LIN {X 0,Y 418.225,Z 378.998,A -85,B 0,C 180,E1 -10215.107,E2 -10215.107} C_VEL
LIN {X 0,Y 418.208,Z 379.016,A -85,B 0,C 180,E1 -10217.763,E2 -10217.763} C_VEL
LIN {X 0,Y 418.223,Z 379.009,A -85,B 0,C 180,E1 -10221.555,E2 -10221.555} C_VEL
LIN {X 0,Y 418.238,Z 379.011,A -85,B 0,C 180,E1 -10225.157,E2 -10225.157} C_VEL
LIN {X 0,Y 418.229,Z 379.012,A -85,B 0,C 180,E1 -10227.471,E2 -10227.471} C_VEL
LIN {X 0,Y 418.247,Z 379.012,A -85,B 0,C 180,E1 -10230.897,E2 -10230.897} C_VEL
LIN {X 0,Y 418.205,Z 379.02,A -85,B 0,C 180,E1 -10234.092,E2 -10234.092} C_VEL
LIN {X 0,Y 418.212,Z 379.016,A -85,B 0,C 180,E1 -10237.263,E2 -10237.263} C_VEL
LIN {X 0,Y 418.236,Z 379.015,A -85,B 0,C 180,E1 -10240.362,E2 -10240.362} C_VEL
LIN {X 0,Y 418.266,Z 379.006,A -85,B 0,C 180,E1 -10243.403,E2 -10243.403} C_VEL
LIN {X 0,Y 418.341,Z 378.997,A -85,B 0,C 180,E1 -10247.385,E2 -10247.385} C_VEL
LIN {X 0,Y 418.311,Z 379,A -85,B 0,C 180,E1 -10250.328,E2 -10250.328} C_VEL
LIN {X 0,Y 418.42,Z 378.982,A -85,B 0,C 180,E1 -10253.248,E2 -10253.248} C_VEL
LIN {X 0,Y 418.301,Z 379.003,A -85,B 0,C 180,E1 -10255.181,E2 -10255.181} C_VEL
LIN {X 0,Y 418.522,Z 378.97,A -85,B 0,C 180,E1 -10258.076,E2 -10258.076} C_VEL
LIN {X 0,Y 418.465,Z 378.979,A -85,B 0,C 180,E1 -10260.963,E2 -10260.963} C_VEL
LIN {X 0,Y 418.46,Z 378.986,A -85,B 0,C 180,E1 -10262.888,E2 -10262.888} C_VEL
LIN {X 0,Y 418.484,Z 378.968,A -85,B 0,C 180,E1 -10265.783,E2 -10265.783} C_VEL
LIN {X 0,Y 418.357,Z 378.985,A -85,B 0,C 180,E1 -10268.696,E2 -10268.696} C_VEL
LIN {X 0,Y 418.298,Z 379.001,A -85,B 0,C 180,E1 -10271.632,E2 -10271.632} C_VEL
LIN {X 0,Y 418.287,Z 378.987,A -85,B 0,C 180,E1 -10274.598,E2 -10274.598} C_VEL
LIN {X 0,Y 418.268,Z 379.006,A -85,B 0,C 180,E1 -10277.605,E2 -10277.605} C_VEL
LIN {X 0,Y 418.238,Z 378.996,A -85,B 0,C 180,E1 -10280.664,E2 -10280.664} C_VEL
LIN {X 0,Y 418.246,Z 379.009,A -85,B 0,C 180,E1 -10283.784,E2 -10283.784} C_VEL
LIN {X 0,Y 418.197,Z 379.005,A -85,B 0,C 180,E1 -10287.044,E2 -10287.044} C_VEL
LIN {X 0,Y 418.23,Z 379.014,A -85,B 0,C 180,E1 -10290.274,E2 -10290.274} C_VEL
LIN {X 0,Y 418.223,Z 379.015,A -85,B 0,C 180,E1 -10293.68,E2 -10293.68} C_VEL
LIN {X 0,Y 418.231,Z 379.009,A -85,B 0,C 180,E1 -10297.226,E2 -10297.226} C_VEL
LIN {X 0,Y 418.203,Z 379.011,A -85,B 0,C 180,E1 -10300.869,E2 -10300.869} C_VEL
LIN {X 0,Y 418.196,Z 379.008,A -85,B 0,C 180,E1 -10303.729,E2 -10303.729} C_VEL
LIN {X 0,Y 418.197,Z 379.016,A -85,B 0,C 180,E1 -10306.449,E2 -10306.449} C_VEL
LIN {X 0,Y 418.206,Z 379.014,A -85,B 0,C 180,E1 -10309.133,E2 -10309.133} C_VEL
LIN {X 0,Y 418.234,Z 379.012,A -85,B 0,C 180,E1 -10312.777,E2 -10312.777} C_VEL
LIN {X 0,Y 418.232,Z 379.027,A -85,B 0,C 180,E1 -10313.708,E2 -10313.708} C_VEL
LIN {X 0,Y 419.156,Z 381.703,A -85,B 0,C 180,E1 -10313.837,E2 -10313.837} C_VEL
LIN {X 0,Y 427.959,Z 397.955,A -85,B 0,C 180,E1 -10314.847,E2 -10314.847} C_VEL
LIN {X 0,Y 431.976,Z 406.121,A -85,B 0,C 180,E1 -10315.304,E2 -10315.304} C_VEL
LIN {X 0,Y 430.27,Z 505.847,A -85,B 0,C 180,E1 -10317.043,E2 -10317.043} C_VEL
LIN {X 0,Y 430.034,Z 520.714,A -85,B 0,C 180,E1 -10317.434,E2 -10317.434} C_VEL
LIN {X 0,Y 429.577,Z 534.376,A -85,B 0,C 180,E1 -10317.957,E2 -10317.957} C_VEL
LIN {X 0,Y 428.77,Z 549.291,A -85,B 0,C 180,E1 -10318.728,E2 -10318.728} C_VEL
LIN {X 0,Y 427.854,Z 563.226,A -85,B 0,C 180,E1 -10319.663,E2 -10319.663} C_VEL
LIN {X 0,Y 426.767,Z 576.005,A -85,B 0,C 180,E1 -10320.72,E2 -10320.72} C_VEL
LIN {X 0,Y 425.445,Z 589.124,A -85,B 0,C 180,E1 -10322.049,E2 -10322.049} C_VEL
LIN {X 0,Y 424.226,Z 600.556,A -85,B 0,C 180,E1 -10323.458,E2 -10323.458} C_VEL
LIN {X 0,Y 423.081,Z 610.61,A -85,B 0,C 180,E1 -10324.94,E2 -10324.94} C_VEL
LIN {X 0,Y 421.854,Z 620.502,A -85,B 0,C 180,E1 -10326.693,E2 -10326.693} C_VEL
LIN {X 0,Y 420.828,Z 628.634,A -85,B 0,C 180,E1 -10328.445,E2 -10328.445} C_VEL
LIN {X 0,Y 419.959,Z 636.143,A -85,B 0,C 180,E1 -10330.447,E2 -10330.447} C_VEL
LIN {X 0,Y 419.257,Z 642.041,A -85,B 0,C 180,E1 -10332.439,E2 -10332.439} C_VEL
LIN {X 0,Y 418.717,Z 646.508,A -85,B 0,C 180,E1 -10334.423,E2 -10334.423} C_VEL
LIN {X 0,Y 418.36,Z 649.659,A -85,B 0,C 180,E1 -10336.398,E2 -10336.398} C_VEL
LIN {X 0,Y 418.275,Z 650.576,A -85,B 0,C 180,E1 -10337.198,E2 -10337.198} C_VEL
LIN {X 0,Y 417.576,Z 651.446,A -85,B 0,C 180,E1 -10337.993,E2 -10337.993} C_VEL
LIN {X 0,Y 414.651,Z 652.693,A -85,B 0,C 180,E1 -10339.286,E2 -10339.286} C_VEL
LIN {X 0,Y 412.192,Z 653.314,A -85,B 0,C 180,E1 -10340.333,E2 -10340.333} C_VEL
LIN {X 0,Y 411.142,Z 653.446,A -85,B 0,C 180,E1 -10341.145,E2 -10341.145} C_VEL
LIN {X 0,Y 411.06,Z 653.387,A -85,B 0,C 180,E1 -10341.421,E2 -10341.421} C_VEL
LIN {X 0,Y 411.156,Z 652.686,A -85,B 0,C 180,E1 -10343.129,E2 -10343.129} C_VEL
LIN {X 0,Y 411.262,Z 651.881,A -85,B 0,C 180,E1 -10344.115,E2 -10344.115} C_VEL
LIN {X 0,Y 411.252,Z 649.436,A -85,B 0,C 180,E1 -10346.081,E2 -10346.081} C_VEL
LIN {X 0,Y 411.645,Z 645.781,A -85,B 0,C 180,E1 -10348.044,E2 -10348.044} C_VEL
LIN {X 0,Y 412.028,Z 640.918,A -85,B 0,C 180,E1 -10350,E2 -10350} C_VEL
LIN {X 0,Y 412.777,Z 634.656,A -85,B 0,C 180,E1 -10351.952,E2 -10351.952} C_VEL
LIN {X 0,Y 413.577,Z 626.87,A -85,B 0,C 180,E1 -10353.898,E2 -10353.898} C_VEL
LIN {X 0,Y 414.448,Z 618.574,A -85,B 0,C 180,E1 -10355.596,E2 -10355.596} C_VEL
LIN {X 0,Y 415.58,Z 608.585,A -85,B 0,C 180,E1 -10357.287,E2 -10357.287} C_VEL
LIN {X 0,Y 416.58,Z 598.393,A -85,B 0,C 180,E1 -10358.733,E2 -10358.733} C_VEL
LIN {X 0,Y 417.615,Z 586.207,A -85,B 0,C 180,E1 -10360.178,E2 -10360.178} C_VEL
LIN {X 0,Y 418.736,Z 573.907,A -85,B 0,C 180,E1 -10361.374,E2 -10361.374} C_VEL
LIN {X 0,Y 419.753,Z 560.42,A -85,B 0,C 180,E1 -10362.449,E2 -10362.449} C_VEL
LIN {X 0,Y 420.664,Z 546.329,A -85,B 0,C 180,E1 -10363.342,E2 -10363.342} C_VEL
LIN {X 0,Y 421.326,Z 532.229,A -85,B 0,C 180,E1 -10364.037,E2 -10364.037} C_VEL
LIN {X 0,Y 421.665,Z 517.374,A -85,B 0,C 180,E1 -10364.578,E2 -10364.578} C_VEL
LIN {X 0,Y 421.841,Z 502.126,A -85,B 0,C 180,E1 -10364.937,E2 -10364.937} C_VEL
LIN {X 0,Y 423.234,Z 406.51,A -85,B 0,C 180,E1 -10366.596,E2 -10366.596} C_VEL
LIN {X 0,Y 412.309,Z 382.923,A -85,B 0,C 180,E1 -10367.72,E2 -10367.72} C_VEL
LIN {X 0,Y 411.343,Z 380.705,A -85,B 0,C 180,E1 -10367.825,E2 -10367.825} C_VEL
LIN {X 0,Y 411.208,Z 379.886,A -85,B 0,C 180,E1 -10367.88,E2 -10367.88} C_VEL
LIN {X 0,Y 411.188,Z 379.894,A -85,B 0,C 180,E1 -10371.034,E2 -10371.034} C_VEL
LIN {X 0,Y 411.172,Z 379.892,A -85,B 0,C 180,E1 -10374.219,E2 -10374.219} C_VEL
LIN {X 0,Y 411.141,Z 379.899,A -85,B 0,C 180,E1 -10377.486,E2 -10377.486} C_VEL
LIN {X 0,Y 411.192,Z 379.876,A -85,B 0,C 180,E1 -10379.713,E2 -10379.713} C_VEL
LIN {X 0,Y 411.202,Z 379.89,A -85,B 0,C 180,E1 -10383.156,E2 -10383.156} C_VEL
LIN {X 0,Y 411.187,Z 379.889,A -85,B 0,C 180,E1 -10386.551,E2 -10386.551} C_VEL
LIN {X 0,Y 411.165,Z 379.887,A -85,B 0,C 180,E1 -10389.719,E2 -10389.719} C_VEL
LIN {X 0,Y 411.115,Z 379.898,A -85,B 0,C 180,E1 -10393.14,E2 -10393.14} C_VEL
LIN {X 0,Y 411.157,Z 379.892,A -85,B 0,C 180,E1 -10395.882,E2 -10395.882} C_VEL
LIN {X 0,Y 411.143,Z 379.894,A -85,B 0,C 180,E1 -10398.774,E2 -10398.774} C_VEL
LIN {X 0,Y 411.177,Z 379.887,A -85,B 0,C 180,E1 -10402.024,E2 -10402.024} C_VEL
LIN {X 0,Y 411.196,Z 379.891,A -85,B 0,C 180,E1 -10405.123,E2 -10405.123} C_VEL
LIN {X 0,Y 411.147,Z 379.894,A -85,B 0,C 180,E1 -10408.001,E2 -10408.001} C_VEL
LIN {X 0,Y 411.161,Z 379.891,A -85,B 0,C 180,E1 -10411.405,E2 -10411.405} C_VEL
LIN {X 0,Y 411.181,Z 379.891,A -85,B 0,C 180,E1 -10414.941,E2 -10414.941} C_VEL
LIN {X 0,Y 411.196,Z 379.888,A -85,B 0,C 180,E1 -10417.913,E2 -10417.913} C_VEL
LIN {X 0,Y 411.211,Z 379.883,A -85,B 0,C 180,E1 -10421.051,E2 -10421.051} C_VEL
LIN {X 0,Y 411.238,Z 379.881,A -85,B 0,C 180,E1 -10424.131,E2 -10424.131} C_VEL
LIN {X 0,Y 411.295,Z 379.862,A -85,B 0,C 180,E1 -10427.165,E2 -10427.165} C_VEL
LIN {X 0,Y 411.27,Z 379.855,A -85,B 0,C 180,E1 -10430.16,E2 -10430.16} C_VEL
LIN {X 0,Y 411.381,Z 379.861,A -85,B 0,C 180,E1 -10433.131,E2 -10433.131} C_VEL
LIN {X 0,Y 411.271,Z 379.88,A -85,B 0,C 180,E1 -10435.098,E2 -10435.098} C_VEL
LIN {X 0,Y 411.488,Z 379.845,A -85,B 0,C 180,E1 -10438.042,E2 -10438.042} C_VEL
LIN {X 0,Y 411.495,Z 379.848,A -85,B 0,C 180,E1 -10441.957,E2 -10441.957} C_VEL
LIN {X 0,Y 411.402,Z 379.864,A -85,B 0,C 180,E1 -10445.883,E2 -10445.883} C_VEL
LIN {X 0,Y 411.299,Z 379.869,A -85,B 0,C 180,E1 -10448.846,E2 -10448.846} C_VEL
LIN {X 0,Y 411.271,Z 379.881,A -85,B 0,C 180,E1 -10451.833,E2 -10451.833} C_VEL
LIN {X 0,Y 411.211,Z 379.88,A -85,B 0,C 180,E1 -10454.854,E2 -10454.854} C_VEL
LIN {X 0,Y 411.169,Z 379.89,A -85,B 0,C 180,E1 -10457.919,E2 -10457.919} C_VEL
LIN {X 0,Y 411.177,Z 379.891,A -85,B 0,C 180,E1 -10461.035,E2 -10461.035} C_VEL
LIN {X 0,Y 411.181,Z 379.891,A -85,B 0,C 180,E1 -10464.218,E2 -10464.218} C_VEL
LIN {X 0,Y 411.139,Z 379.896,A -85,B 0,C 180,E1 -10467.486,E2 -10467.486} C_VEL
LIN {X 0,Y 411.188,Z 379.891,A -85,B 0,C 180,E1 -10469.713,E2 -10469.713} C_VEL
LIN {X 0,Y 411.197,Z 379.883,A -85,B 0,C 180,E1 -10473.156,E2 -10473.156} C_VEL
LIN {X 0,Y 411.181,Z 379.891,A -85,B 0,C 180,E1 -10476.552,E2 -10476.552} C_VEL
LIN {X 0,Y 411.161,Z 379.891,A -85,B 0,C 180,E1 -10479.72,E2 -10479.72} C_VEL
LIN {X 0,Y 411.156,Z 379.89,A -85,B 0,C 180,E1 -10483.136,E2 -10483.136} C_VEL
LIN {X 0,Y 411.158,Z 379.891,A -85,B 0,C 180,E1 -10485.882,E2 -10485.882} C_VEL
LIN {X 0,Y 411.141,Z 379.88,A -85,B 0,C 180,E1 -10488.775,E2 -10488.775} C_VEL
LIN {X 0,Y 411.191,Z 379.892,A -85,B 0,C 180,E1 -10492.304,E2 -10492.304} C_VEL
LIN {X 0,Y 411.198,Z 380.027,A -85,B 0,C 180,E1 -10492.444,E2 -10492.444} C_VEL
LIN {X 0,Y 416.322,Z 398.71,A -85,B 0,C 180,E1 -10495.433,E2 -10495.433} C_VEL
LIN {X 0,Y 419.282,Z 410.864,A -85,B 0,C 180,E1 -10497.271,E2 -10497.271} C_VEL
LIN {X 0,Y 418.63,Z 422.432,A -85,B 0,C 180,E1 -10498.783,E2 -10498.783} C_VEL
LIN {X 0,Y 416.677,Z 449.268,A -85,B 0,C 180,E1 -10502.229,E2 -10502.229} C_VEL
LIN {X 0,Y 416.403,Z 453.768,A -85,B 0,C 180,E1 -10502.805,E2 -10502.805} C_VEL
LIN {X 0,Y 422.661,Z 500.014,A -85,B 0,C 180,E1 -10504.019,E2 -10504.019} C_VEL
LIN {X 0,Y 420.619,Z 622.26,A -85,B 0,C 180,E1 -10506.13,E2 -10506.13} C_VEL
LIN {X 0,Y 419.884,Z 638.091,A -85,B 0,C 180,E1 -10506.577,E2 -10506.577} C_VEL
LIN {X 0,Y 418.756,Z 653.905,A -85,B 0,C 180,E1 -10507.229,E2 -10507.229} C_VEL
LIN {X 0,Y 417.474,Z 669.239,A -85,B 0,C 180,E1 -10508.087,E2 -10508.087} C_VEL
LIN {X 0,Y 416.242,Z 683.405,A -85,B 0,C 180,E1 -10509.104,E2 -10509.104} C_VEL
LIN {X 0,Y 414.909,Z 697.181,A -85,B 0,C 180,E1 -10510.327,E2 -10510.327} C_VEL
LIN {X 0,Y 413.738,Z 709.762,A -85,B 0,C 180,E1 -10511.684,E2 -10511.684} C_VEL
LIN {X 0,Y 412.662,Z 721.262,A -85,B 0,C 180,E1 -10513.171,E2 -10513.171} C_VEL
LIN {X 0,Y 411.697,Z 732.447,A -85,B 0,C 180,E1 -10514.91,E2 -10514.91} C_VEL
LIN {X 0,Y 411.075,Z 741.798,A -85,B 0,C 180,E1 -10516.656,E2 -10516.656} C_VEL
LIN {X 0,Y 410.666,Z 750.567,A -85,B 0,C 180,E1 -10518.65,E2 -10518.65} C_VEL
LIN {X 0,Y 410.452,Z 757.62,A -85,B 0,C 180,E1 -10520.638,E2 -10520.638} C_VEL
LIN {X 0,Y 410.492,Z 763.175,A -85,B 0,C 180,E1 -10522.622,E2 -10522.622} C_VEL
LIN {X 0,Y 410.534,Z 766.369,A -85,B 0,C 180,E1 -10524.104,E2 -10524.104} C_VEL
LIN {X 0,Y 410.65,Z 769.529,A -85,B 0,C 180,E1 -10526.074,E2 -10526.074} C_VEL
LIN {X 0,Y 410.673,Z 771.422,A -85,B 0,C 180,E1 -10528.038,E2 -10528.038} C_VEL
LIN {X 0,Y 410.871,Z 771.932,A -85,B 0,C 180,E1 -10529.02,E2 -10529.02} C_VEL
LIN {X 0,Y 410.871,Z 771.945,A -85,B 0,C 180,E1 -10530.98,E2 -10530.98} C_VEL
LIN {X 0,Y 410.647,Z 770.73,A -85,B 0,C 180,E1 -10532.943,E2 -10532.943} C_VEL
LIN {X 0,Y 410.624,Z 768.339,A -85,B 0,C 180,E1 -10534.909,E2 -10534.909} C_VEL
LIN {X 0,Y 410.537,Z 764.69,A -85,B 0,C 180,E1 -10536.882,E2 -10536.882} C_VEL
LIN {X 0,Y 410.42,Z 759.703,A -85,B 0,C 180,E1 -10538.865,E2 -10538.865} C_VEL
LIN {X 0,Y 410.591,Z 753.288,A -85,B 0,C 180,E1 -10540.852,E2 -10540.852} C_VEL
LIN {X 0,Y 410.918,Z 745.181,A -85,B 0,C 180,E1 -10542.87,E2 -10542.87} C_VEL
LIN {X 0,Y 411.528,Z 736.805,A -85,B 0,C 180,E1 -10544.589,E2 -10544.589} C_VEL
LIN {X 0,Y 412.413,Z 726.708,A -85,B 0,C 180,E1 -10546.33,E2 -10546.33} C_VEL
LIN {X 0,Y 413.445,Z 716.287,A -85,B 0,C 180,E1 -10547.839,E2 -10547.839} C_VEL
LIN {X 0,Y 414.704,Z 704.353,A -85,B 0,C 180,E1 -10549.296,E2 -10549.296} C_VEL
LIN {X 0,Y 416.107,Z 691.061,A -85,B 0,C 180,E1 -10550.644,E2 -10550.644} C_VEL
LIN {X 0,Y 417.599,Z 677.926,A -85,B 0,C 180,E1 -10551.73,E2 -10551.73} C_VEL
LIN {X 0,Y 418.974,Z 663.594,A -85,B 0,C 180,E1 -10552.693,E2 -10552.693} C_VEL
LIN {X 0,Y 420.373,Z 648.783,A -85,B 0,C 180,E1 -10553.459,E2 -10553.459} C_VEL
LIN {X 0,Y 421.533,Z 633.428,A -85,B 0,C 180,E1 -10554.043,E2 -10554.043} C_VEL
LIN {X 0,Y 422.265,Z 618.692,A -85,B 0,C 180,E1 -10554.423,E2 -10554.423} C_VEL
LIN {X 0,Y 424.406,Z 499.375,A -85,B 0,C 180,E1 -10556.522,E2 -10556.522} C_VEL
LIN {X 0,Y 420.436,Z 470.006,A -85,B 0,C 180,E1 -10557.373,E2 -10557.373} C_VEL
LIN {X 0,Y 417.477,Z 452.12,A -85,B 0,C 180,E1 -10557.966,E2 -10557.966} C_VEL
LIN {X 0,Y 419.58,Z 426.838,A -85,B 0,C 180,E1 -10561.323,E2 -10561.323} C_VEL
LIN {X 0,Y 420.768,Z 414.209,A -85,B 0,C 180,E1 -10563.018,E2 -10563.018} C_VEL
LIN {X 0,Y 417.56,Z 401.012,A -85,B 0,C 180,E1 -10565.175,E2 -10565.175} C_VEL
LIN {X 0,Y 412.955,Z 385.69,A -85,B 0,C 180,E1 -10567.889,E2 -10567.889} C_VEL
LIN {X 0,Y 411.169,Z 379.895,A -85,B 0,C 180,E1 -10568.971,E2 -10568.971} C_VEL
LIN {X 0,Y 411.158,Z 379.891,A -85,B 0,C 180,E1 -10572.693,E2 -10572.693} C_VEL
LIN {X 0,Y 411.153,Z 379.878,A -85,B 0,C 180,E1 -10575.881,E2 -10575.881} C_VEL
LIN {X 0,Y 411.147,Z 379.893,A -85,B 0,C 180,E1 -10579.492,E2 -10579.492} C_VEL
LIN {X 0,Y 411.17,Z 379.891,A -85,B 0,C 180,E1 -10582.024,E2 -10582.024} C_VEL
LIN {X 0,Y 411.19,Z 379.89,A -85,B 0,C 180,E1 -10585.123,E2 -10585.123} C_VEL
LIN {X 0,Y 411.151,Z 379.897,A -85,B 0,C 180,E1 -10588.002,E2 -10588.002} C_VEL
LIN {X 0,Y 411.159,Z 379.894,A -85,B 0,C 180,E1 -10591.406,E2 -10591.406} C_VEL
LIN {X 0,Y 411.175,Z 379.89,A -85,B 0,C 180,E1 -10594.941,E2 -10594.941} C_VEL
LIN {X 0,Y 411.185,Z 379.893,A -85,B 0,C 180,E1 -10597.913,E2 -10597.913} C_VEL
LIN {X 0,Y 411.168,Z 379.893,A -85,B 0,C 180,E1 -10601.049,E2 -10601.049} C_VEL
LIN {X 0,Y 411.194,Z 379.891,A -85,B 0,C 180,E1 -10604.13,E2 -10604.13} C_VEL
LIN {X 0,Y 411.289,Z 379.877,A -85,B 0,C 180,E1 -10607.165,E2 -10607.165} C_VEL
LIN {X 0,Y 411.266,Z 379.877,A -85,B 0,C 180,E1 -10610.161,E2 -10610.161} C_VEL
LIN {X 0,Y 411.371,Z 379.861,A -85,B 0,C 180,E1 -10613.132,E2 -10613.132} C_VEL
LIN {X 0,Y 411.272,Z 379.879,A -85,B 0,C 180,E1 -10615.099,E2 -10615.099} C_VEL
LIN {X 0,Y 411.491,Z 379.846,A -85,B 0,C 180,E1 -10618.043,E2 -10618.043} C_VEL
LIN {X 0,Y 411.488,Z 379.847,A -85,B 0,C 180,E1 -10621.958,E2 -10621.958} C_VEL
LIN {X 0,Y 411.429,Z 379.846,A -85,B 0,C 180,E1 -10625.883,E2 -10625.883} C_VEL
LIN {X 0,Y 411.4,Z 379.843,A -85,B 0,C 180,E1 -10627.855,E2 -10627.855} C_VEL
LIN {X 0,Y 411.268,Z 379.877,A -85,B 0,C 180,E1 -10631.833,E2 -10631.833} C_VEL
LIN {X 0,Y 411.245,Z 379.865,A -85,B 0,C 180,E1 -10634.854,E2 -10634.854} C_VEL
LIN {X 0,Y 411.233,Z 379.882,A -85,B 0,C 180,E1 -10637.916,E2 -10637.916} C_VEL
LIN {X 0,Y 411.184,Z 379.874,A -85,B 0,C 180,E1 -10641.035,E2 -10641.035} C_VEL
LIN {X 0,Y 411.18,Z 379.891,A -85,B 0,C 180,E1 -10644.219,E2 -10644.219} C_VEL
LIN {X 0,Y 411.138,Z 379.887,A -85,B 0,C 180,E1 -10647.487,E2 -10647.487} C_VEL
LIN {X 0,Y 411.187,Z 379.891,A -85,B 0,C 180,E1 -10649.714,E2 -10649.714} C_VEL
LIN {X 0,Y 411.195,Z 379.886,A -85,B 0,C 180,E1 -10653.157,E2 -10653.157} C_VEL
LIN {X 0,Y 411.184,Z 379.884,A -85,B 0,C 180,E1 -10656.553,E2 -10656.553} C_VEL
LIN {X 0,Y 411.17,Z 379.889,A -85,B 0,C 180,E1 -10659.723,E2 -10659.723} C_VEL
LIN {X 0,Y 411.156,Z 379.89,A -85,B 0,C 180,E1 -10663.136,E2 -10663.136} C_VEL
LIN {X 0,Y 411.159,Z 379.893,A -85,B 0,C 180,E1 -10665.883,E2 -10665.883} C_VEL
LIN {X 0,Y 411.146,Z 379.897,A -85,B 0,C 180,E1 -10668.775,E2 -10668.775} C_VEL
LIN {X 0,Y 411.183,Z 379.886,A -85,B 0,C 180,E1 -10672.027,E2 -10672.027} C_VEL
LIN {X 0,Y 411.175,Z 379.926,A -85,B 0,C 180,E1 -10673.132,E2 -10673.132} C_VEL
LIN {X 0,Y 412.271,Z 382.902,A -85,B 0,C 180,E1 -10673.286,E2 -10673.286} C_VEL
LIN {X 0,Y 418.282,Z 393.569,A -85,B 0,C 180,E1 -10673.998,E2 -10673.998} C_VEL
LIN {X 0,Y 425.769,Z 408.425,A -85,B 0,C 180,E1 -10674.878,E2 -10674.878} C_VEL
LIN {X 0,Y 424.008,Z 504.93,A -85,B 0,C 180,E1 -10676.578,E2 -10676.578} C_VEL
LIN {X 0,Y 423.778,Z 520.195,A -85,B 0,C 180,E1 -10676.963,E2 -10676.963} C_VEL
LIN {X 0,Y 423.244,Z 535.512,A -85,B 0,C 180,E1 -10677.552,E2 -10677.552} C_VEL
LIN {X 0,Y 422.458,Z 549.577,A -85,B 0,C 180,E1 -10678.284,E2 -10678.284} C_VEL
LIN {X 0,Y 421.551,Z 562.682,A -85,B 0,C 180,E1 -10679.16,E2 -10679.16} C_VEL
LIN {X 0,Y 420.463,Z 575.265,A -85,B 0,C 180,E1 -10680.193,E2 -10680.193} C_VEL
LIN {X 0,Y 419.158,Z 587.941,A -85,B 0,C 180,E1 -10681.456,E2 -10681.456} C_VEL
LIN {X 0,Y 417.988,Z 598.56,A -85,B 0,C 180,E1 -10682.732,E2 -10682.732} C_VEL
LIN {X 0,Y 416.703,Z 609.258,A -85,B 0,C 180,E1 -10684.261,E2 -10684.261} C_VEL
LIN {X 0,Y 415.338,Z 619.516,A -85,B 0,C 180,E1 -10686.028,E2 -10686.028} C_VEL
LIN {X 0,Y 414.23,Z 628.044,A -85,B 0,C 180,E1 -10687.822,E2 -10687.822} C_VEL
LIN {X 0,Y 413.329,Z 635.134,A -85,B 0,C 180,E1 -10689.64,E2 -10689.64} C_VEL
LIN {X 0,Y 412.543,Z 641.369,A -85,B 0,C 180,E1 -10691.63,E2 -10691.63} C_VEL
LIN {X 0,Y 411.907,Z 646.26,A -85,B 0,C 180,E1 -10693.65,E2 -10693.65} C_VEL
LIN {X 0,Y 411.573,Z 649.057,A -85,B 0,C 180,E1 -10695.16,E2 -10695.16} C_VEL
LIN {X 0,Y 411.289,Z 651.669,A -85,B 0,C 180,E1 -10697.166,E2 -10697.166} C_VEL
LIN {X 0,Y 411.107,Z 653.122,A -85,B 0,C 180,E1 -10699.162,E2 -10699.162} C_VEL
LIN {X 0,Y 411.06,Z 653.387,A -85,B 0,C 180,E1 -10701.421,E2 -10701.421} C_VEL
LIN {X 0,Y 410.407,Z 653.267,A -85,B 0,C 180,E1 -10702.239,E2 -10702.239} C_VEL
LIN {X 0,Y 407.587,Z 652.849,A -85,B 0,C 180,E1 -10703.571,E2 -10703.571} C_VEL
LIN {X 0,Y 405.227,Z 652.195,A -85,B 0,C 180,E1 -10704.642,E2 -10704.642} C_VEL
LIN {X 0,Y 404.251,Z 651.376,A -85,B 0,C 180,E1 -10705.464,E2 -10705.464} C_VEL
LIN {X 0,Y 404.192,Z 650.978,A -85,B 0,C 180,E1 -10705.74,E2 -10705.74} C_VEL
LIN {X 0,Y 404.477,Z 648.958,A -85,B 0,C 180,E1 -10707.012,E2 -10707.012} C_VEL
LIN {X 0,Y 404.753,Z 644.808,A -85,B 0,C 180,E1 -10709.005,E2 -10709.005} C_VEL
LIN {X 0,Y 405.383,Z 639.336,A -85,B 0,C 180,E1 -10710.994,E2 -10710.994} C_VEL
LIN {X 0,Y 406.195,Z 632.424,A -85,B 0,C 180,E1 -10712.976,E2 -10712.976} C_VEL
LIN {X 0,Y 407.11,Z 623.87,A -85,B 0,C 180,E1 -10714.952,E2 -10714.952} C_VEL
LIN {X 0,Y 408.172,Z 614.756,A -85,B 0,C 180,E1 -10716.674,E2 -10716.674} C_VEL
LIN {X 0,Y 409.362,Z 603.78,A -85,B 0,C 180,E1 -10718.391,E2 -10718.391} C_VEL
LIN {X 0,Y 410.492,Z 592.459,A -85,B 0,C 180,E1 -10719.858,E2 -10719.858} C_VEL
LIN {X 0,Y 411.441,Z 581.251,A -85,B 0,C 180,E1 -10721.079,E2 -10721.079} C_VEL
LIN {X 0,Y 412.547,Z 569.151,A -85,B 0,C 180,E1 -10722.17,E2 -10722.17} C_VEL
LIN {X 0,Y 413.496,Z 556.081,A -85,B 0,C 180,E1 -10723.14,E2 -10723.14} C_VEL
LIN {X 0,Y 414.348,Z 541.609,A -85,B 0,C 180,E1 -10723.986,E2 -10723.986} C_VEL
LIN {X 0,Y 414.941,Z 526.466,A -85,B 0,C 180,E1 -10724.654,E2 -10724.654} C_VEL
LIN {X 0,Y 415.216,Z 510.775,A -85,B 0,C 180,E1 -10725.133,E2 -10725.133} C_VEL
LIN {X 0,Y 416.29,Z 438.184,A -85,B 0,C 180,E1 -10726.434,E2 -10726.434} C_VEL
LIN {X 0,Y 416.69,Z 408.385,A -85,B 0,C 180,E1 -10726.963,E2 -10726.963} C_VEL
LIN {X 0,Y 406.217,Z 385.8,A -85,B 0,C 180,E1 -10728.067,E2 -10728.067} C_VEL
LIN {X 0,Y 404.264,Z 381.548,A -85,B 0,C 180,E1 -10728.281,E2 -10728.281} C_VEL
LIN {X 0,Y 404.124,Z 380.77,A -85,B 0,C 180,E1 -10728.308,E2 -10728.308} C_VEL
LIN {X 0,Y 404.132,Z 380.77,A -85,B 0,C 180,E1 -10731.42,E2 -10731.42} C_VEL
LIN {X 0,Y 404.128,Z 380.771,A -85,B 0,C 180,E1 -10734.669,E2 -10734.669} C_VEL
LIN {X 0,Y 404.099,Z 380.774,A -85,B 0,C 180,E1 -10738.006,E2 -10738.006} C_VEL
LIN {X 0,Y 404.139,Z 380.754,A -85,B 0,C 180,E1 -10740.285,E2 -10740.285} C_VEL
LIN {X 0,Y 404.135,Z 380.765,A -85,B 0,C 180,E1 -10743.813,E2 -10743.813} C_VEL
LIN {X 0,Y 404.129,Z 380.768,A -85,B 0,C 180,E1 -10746.873,E2 -10746.873} C_VEL
LIN {X 0,Y 404.115,Z 380.764,A -85,B 0,C 180,E1 -10750.074,E2 -10750.074} C_VEL
LIN {X 0,Y 404.074,Z 380.775,A -85,B 0,C 180,E1 -10753.071,E2 -10753.071} C_VEL
LIN {X 0,Y 404.114,Z 380.769,A -85,B 0,C 180,E1 -10755.921,E2 -10755.921} C_VEL
LIN {X 0,Y 404.097,Z 380.77,A -85,B 0,C 180,E1 -10758.632,E2 -10758.632} C_VEL
LIN {X 0,Y 404.133,Z 380.766,A -85,B 0,C 180,E1 -10761.495,E2 -10761.495} C_VEL
LIN {X 0,Y 404.167,Z 380.767,A -85,B 0,C 180,E1 -10764.982,E2 -10764.982} C_VEL
LIN {X 0,Y 404.124,Z 380.769,A -85,B 0,C 180,E1 -10768.444,E2 -10768.444} C_VEL
LIN {X 0,Y 404.141,Z 380.765,A -85,B 0,C 180,E1 -10770.861,E2 -10770.861} C_VEL
LIN {X 0,Y 404.145,Z 380.766,A -85,B 0,C 180,E1 -10774.723,E2 -10774.723} C_VEL
LIN {X 0,Y 404.159,Z 380.767,A -85,B 0,C 180,E1 -10777.507,E2 -10777.507} C_VEL
LIN {X 0,Y 404.154,Z 380.761,A -85,B 0,C 180,E1 -10780.707,E2 -10780.707} C_VEL
LIN {X 0,Y 404.209,Z 380.759,A -85,B 0,C 180,E1 -10783.847,E2 -10783.847} C_VEL
LIN {X 0,Y 404.276,Z 380.74,A -85,B 0,C 180,E1 -10786.938,E2 -10786.938} C_VEL
LIN {X 0,Y 404.237,Z 380.728,A -85,B 0,C 180,E1 -10789.988,E2 -10789.988} C_VEL
LIN {X 0,Y 404.332,Z 380.738,A -85,B 0,C 180,E1 -10793.011,E2 -10793.011} C_VEL
LIN {X 0,Y 404.243,Z 380.755,A -85,B 0,C 180,E1 -10795.013,E2 -10795.013} C_VEL
LIN {X 0,Y 404.457,Z 380.72,A -85,B 0,C 180,E1 -10798.008,E2 -10798.008} C_VEL
LIN {X 0,Y 404.464,Z 380.723,A -85,B 0,C 180,E1 -10801.991,E2 -10801.991} C_VEL
LIN {X 0,Y 404.352,Z 380.741,A -85,B 0,C 180,E1 -10805.986,E2 -10805.986} C_VEL
LIN {X 0,Y 404.248,Z 380.748,A -85,B 0,C 180,E1 -10809.002,E2 -10809.002} C_VEL
LIN {X 0,Y 404.245,Z 380.754,A -85,B 0,C 180,E1 -10812.042,E2 -10812.042} C_VEL
LIN {X 0,Y 404.159,Z 380.759,A -85,B 0,C 180,E1 -10815.12,E2 -10815.12} C_VEL
LIN {X 0,Y 404.126,Z 380.764,A -85,B 0,C 180,E1 -10818.242,E2 -10818.242} C_VEL
LIN {X 0,Y 404.122,Z 380.773,A -85,B 0,C 180,E1 -10821.42,E2 -10821.42} C_VEL
LIN {X 0,Y 404.127,Z 380.768,A -85,B 0,C 180,E1 -10824.669,E2 -10824.669} C_VEL
LIN {X 0,Y 404.096,Z 380.775,A -85,B 0,C 180,E1 -10828.007,E2 -10828.007} C_VEL
LIN {X 0,Y 404.135,Z 380.77,A -85,B 0,C 180,E1 -10830.286,E2 -10830.286} C_VEL
LIN {X 0,Y 404.131,Z 380.76,A -85,B 0,C 180,E1 -10833.813,E2 -10833.813} C_VEL
LIN {X 0,Y 404.124,Z 380.77,A -85,B 0,C 180,E1 -10836.874,E2 -10836.874} C_VEL
LIN {X 0,Y 404.111,Z 380.775,A -85,B 0,C 180,E1 -10840.075,E2 -10840.075} C_VEL
LIN {X 0,Y 404.135,Z 380.764,A -85,B 0,C 180,E1 -10843.082,E2 -10843.082} C_VEL
LIN {X 0,Y 404.115,Z 380.768,A -85,B 0,C 180,E1 -10845.922,E2 -10845.922} C_VEL
LIN {X 0,Y 404.095,Z 380.758,A -85,B 0,C 180,E1 -10848.633,E2 -10848.633} C_VEL
LIN {X 0,Y 404.134,Z 380.808,A -85,B 0,C 180,E1 -10852.02,E2 -10852.02} C_VEL
LIN {X 0,Y 409.274,Z 399.503,A -85,B 0,C 180,E1 -10855.08,E2 -10855.08} C_VEL
LIN {X 0,Y 412.489,Z 412.631,A -85,B 0,C 180,E1 -10857.107,E2 -10857.107} C_VEL
LIN {X 0,Y 411.815,Z 423.657,A -85,B 0,C 180,E1 -10858.572,E2 -10858.572} C_VEL
LIN {X 0,Y 409.865,Z 448.871,A -85,B 0,C 180,E1 -10861.866,E2 -10861.866} C_VEL
LIN {X 0,Y 409.658,Z 453.015,A -85,B 0,C 180,E1 -10862.38,E2 -10862.38} C_VEL
LIN {X 0,Y 416.102,Z 500.849,A -85,B 0,C 180,E1 -10863.659,E2 -10863.659} C_VEL
LIN {X 0,Y 414.038,Z 619.207,A -85,B 0,C 180,E1 -10865.727,E2 -10865.727} C_VEL
LIN {X 0,Y 413.397,Z 634.93,A -85,B 0,C 180,E1 -10866.153,E2 -10866.153} C_VEL
LIN {X 0,Y 412.38,Z 649.401,A -85,B 0,C 180,E1 -10866.723,E2 -10866.723} C_VEL
LIN {X 0,Y 411.091,Z 664.503,A -85,B 0,C 180,E1 -10867.525,E2 -10867.525} C_VEL
LIN {X 0,Y 409.814,Z 678.67,A -85,B 0,C 180,E1 -10868.496,E2 -10868.496} C_VEL
LIN {X 0,Y 408.507,Z 691.827,A -85,B 0,C 180,E1 -10869.612,E2 -10869.612} C_VEL
LIN {X 0,Y 407.313,Z 704.034,A -85,B 0,C 180,E1 -10870.863,E2 -10870.863} C_VEL
LIN {X 0,Y 406.174,Z 715.18,A -85,B 0,C 180,E1 -10872.219,E2 -10872.219} C_VEL
LIN {X 0,Y 405.256,Z 725.036,A -85,B 0,C 180,E1 -10873.632,E2 -10873.632} C_VEL
LIN {X 0,Y 404.38,Z 735.436,A -85,B 0,C 180,E1 -10875.404,E2 -10875.404} C_VEL
LIN {X 0,Y 403.788,Z 744.341,A -85,B 0,C 180,E1 -10877.233,E2 -10877.233} C_VEL
LIN {X 0,Y 403.57,Z 751.31,A -85,B 0,C 180,E1 -10878.956,E2 -10878.956} C_VEL
LIN {X 0,Y 403.388,Z 757.997,A -85,B 0,C 180,E1 -10880.979,E2 -10880.979} C_VEL
LIN {X 0,Y 403.483,Z 763.533,A -85,B 0,C 180,E1 -10883.14,E2 -10883.14} C_VEL
LIN {X 0,Y 403.567,Z 767.046,A -85,B 0,C 180,E1 -10885.004,E2 -10885.004} C_VEL
LIN {X 0,Y 403.621,Z 769.586,A -85,B 0,C 180,E1 -10887.005,E2 -10887.005} C_VEL
LIN {X 0,Y 403.847,Z 770.904,A -85,B 0,C 180,E1 -10889.002,E2 -10889.002} C_VEL
LIN {X 0,Y 403.846,Z 770.933,A -85,B 0,C 180,E1 -10890.997,E2 -10890.997} C_VEL
LIN {X 0,Y 403.606,Z 769.734,A -85,B 0,C 180,E1 -10892.994,E2 -10892.994} C_VEL
LIN {X 0,Y 403.574,Z 767.36,A -85,B 0,C 180,E1 -10894.995,E2 -10894.995} C_VEL
LIN {X 0,Y 403.451,Z 763.725,A -85,B 0,C 180,E1 -10897.003,E2 -10897.003} C_VEL
LIN {X 0,Y 403.352,Z 758.758,A -85,B 0,C 180,E1 -10899.021,E2 -10899.021} C_VEL
LIN {X 0,Y 403.511,Z 752.356,A -85,B 0,C 180,E1 -10901.045,E2 -10901.045} C_VEL
LIN {X 0,Y 403.885,Z 744.389,A -85,B 0,C 180,E1 -10903.073,E2 -10903.073} C_VEL
LIN {X 0,Y 404.532,Z 735.937,A -85,B 0,C 180,E1 -10904.847,E2 -10904.847} C_VEL
LIN {X 0,Y 405.488,Z 725.884,A -85,B 0,C 180,E1 -10906.617,E2 -10906.617} C_VEL
LIN {X 0,Y 406.567,Z 715.682,A -85,B 0,C 180,E1 -10908.128,E2 -10908.128} C_VEL
LIN {X 0,Y 407.928,Z 703.648,A -85,B 0,C 180,E1 -10909.63,E2 -10909.63} C_VEL
LIN {X 0,Y 409.411,Z 690.435,A -85,B 0,C 180,E1 -10910.997,E2 -10910.997} C_VEL
LIN {X 0,Y 410.962,Z 677.405,A -85,B 0,C 180,E1 -10912.099,E2 -10912.099} C_VEL
LIN {X 0,Y 412.416,Z 663.218,A -85,B 0,C 180,E1 -10913.074,E2 -10913.074} C_VEL
LIN {X 0,Y 413.865,Z 648.623,A -85,B 0,C 180,E1 -10913.851,E2 -10913.851} C_VEL
LIN {X 0,Y 415.104,Z 632.726,A -85,B 0,C 180,E1 -10914.472,E2 -10914.472} C_VEL
LIN {X 0,Y 415.933,Z 616.725,A -85,B 0,C 180,E1 -10914.887,E2 -10914.887} C_VEL
LIN {X 0,Y 418.15,Z 500.316,A -85,B 0,C 180,E1 -10916.961,E2 -10916.961} C_VEL
LIN {X 0,Y 414.373,Z 472.005,A -85,B 0,C 180,E1 -10917.798,E2 -10917.798} C_VEL
LIN {X 0,Y 410.908,Z 451.051,A -85,B 0,C 180,E1 -10918.502,E2 -10918.502} C_VEL
LIN {X 0,Y 413.083,Z 426.468,A -85,B 0,C 180,E1 -10921.83,E2 -10921.83} C_VEL
LIN {X 0,Y 414.066,Z 416.029,A -85,B 0,C 180,E1 -10923.259,E2 -10923.259} C_VEL
LIN {X 0,Y 410.704,Z 402.187,A -85,B 0,C 180,E1 -10925.576,E2 -10925.576} C_VEL
LIN {X 0,Y 405.914,Z 386.579,A -85,B 0,C 180,E1 -10928.423,E2 -10928.423} C_VEL
LIN {X 0,Y 404.138,Z 380.768,A -85,B 0,C 180,E1 -10929.577,E2 -10929.577} C_VEL
LIN {X 0,Y 404.134,Z 380.767,A -85,B 0,C 180,E1 -10933.081,E2 -10933.081} C_VEL
LIN {X 0,Y 404.11,Z 380.755,A -85,B 0,C 180,E1 -10935.921,E2 -10935.921} C_VEL
LIN {X 0,Y 404.091,Z 380.771,A -85,B 0,C 180,E1 -10938.632,E2 -10938.632} C_VEL
LIN {X 0,Y 404.126,Z 380.764,A -85,B 0,C 180,E1 -10941.495,E2 -10941.495} C_VEL
LIN {X 0,Y 404.161,Z 380.766,A -85,B 0,C 180,E1 -10944.982,E2 -10944.982} C_VEL
LIN {X 0,Y 404.125,Z 380.771,A -85,B 0,C 180,E1 -10948.442,E2 -10948.442} C_VEL
LIN {X 0,Y 404.137,Z 380.771,A -85,B 0,C 180,E1 -10950.862,E2 -10950.862} C_VEL
LIN {X 0,Y 404.14,Z 380.769,A -85,B 0,C 180,E1 -10954.722,E2 -10954.722} C_VEL
LIN {X 0,Y 404.15,Z 380.768,A -85,B 0,C 180,E1 -10957.507,E2 -10957.507} C_VEL
LIN {X 0,Y 404.12,Z 380.774,A -85,B 0,C 180,E1 -10960.706,E2 -10960.706} C_VEL
LIN {X 0,Y 404.165,Z 380.764,A -85,B 0,C 180,E1 -10963.846,E2 -10963.846} C_VEL
LIN {X 0,Y 404.27,Z 380.752,A -85,B 0,C 180,E1 -10966.939,E2 -10966.939} C_VEL
LIN {X 0,Y 404.233,Z 380.752,A -85,B 0,C 180,E1 -10969.988,E2 -10969.988} C_VEL
LIN {X 0,Y 404.322,Z 380.739,A -85,B 0,C 180,E1 -10973.011,E2 -10973.011} C_VEL
LIN {X 0,Y 404.243,Z 380.755,A -85,B 0,C 180,E1 -10975.013,E2 -10975.013} C_VEL
LIN {X 0,Y 404.46,Z 380.721,A -85,B 0,C 180,E1 -10978.009,E2 -10978.009} C_VEL
LIN {X 0,Y 404.457,Z 380.723,A -85,B 0,C 180,E1 -10981.992,E2 -10981.992} C_VEL
LIN {X 0,Y 404.359,Z 380.716,A -85,B 0,C 180,E1 -10986.71,E2 -10986.71} C_VEL
LIN {X 0,Y 404.237,Z 380.752,A -85,B 0,C 180,E1 -10990.012,E2 -10990.012} C_VEL
LIN {X 0,Y 404.255,Z 380.737,A -85,B 0,C 180,E1 -10993.212,E2 -10993.212} C_VEL
LIN {X 0,Y 404.205,Z 380.762,A -85,B 0,C 180,E1 -10997.008,E2 -10997.008} C_VEL
LIN {X 0,Y 404.153,Z 380.751,A -85,B 0,C 180,E1 -11000.352,E2 -11000.352} C_VEL
LIN {X 0,Y 404.138,Z 380.767,A -85,B 0,C 180,E1 -11003.577,E2 -11003.577} C_VEL
LIN {X 0,Y 404.093,Z 380.76,A -85,B 0,C 180,E1 -11006.885,E2 -11006.885} C_VEL
LIN {X 0,Y 404.134,Z 380.771,A -85,B 0,C 180,E1 -11010.286,E2 -11010.286} C_VEL
LIN {X 0,Y 404.129,Z 380.77,A -85,B 0,C 180,E1 -11013.814,E2 -11013.814} C_VEL
LIN {X 0,Y 404.127,Z 380.763,A -85,B 0,C 180,E1 -11016.876,E2 -11016.876} C_VEL
LIN {X 0,Y 404.109,Z 380.768,A -85,B 0,C 180,E1 -11020.076,E2 -11020.076} C_VEL
LIN {X 0,Y 404.135,Z 380.765,A -85,B 0,C 180,E1 -11023.083,E2 -11023.083} C_VEL
LIN {X 0,Y 404.14,Z 380.767,A -85,B 0,C 180,E1 -11025.927,E2 -11025.927} C_VEL
LIN {X 0,Y 404.101,Z 380.776,A -85,B 0,C 180,E1 -11028.634,E2 -11028.634} C_VEL
LIN {X 0,Y 404.137,Z 380.766,A -85,B 0,C 180,E1 -11031.496,E2 -11031.496} C_VEL
LIN {X 0,Y 404.133,Z 380.766,A -85,B 0,C 180,E1 -11032.509,E2 -11032.509} C_VEL
LIN {X 0,Y 405.199,Z 383.713,A -85,B 0,C 180,E1 -11032.686,E2 -11032.686} C_VEL
LIN {X 0,Y 406.636,Z 386.162,A -85,B 0,C 180,E1 -11032.863,E2 -11032.863} C_VEL
LIN {X 0,Y 414.899,Z 401.202,A -85,B 0,C 180,E1 -11033.871,E2 -11033.871} C_VEL
LIN {X 0,Y 419.601,Z 410.533,A -85,B 0,C 180,E1 -11034.436,E2 -11034.436} C_VEL
LIN {X 0,Y 417.741,Z 506.376,A -85,B 0,C 180,E1 -11036.148,E2 -11036.148} C_VEL
LIN {X 0,Y 417.498,Z 521.631,A -85,B 0,C 180,E1 -11036.545,E2 -11036.545} C_VEL
LIN {X 0,Y 417.016,Z 535.396,A -85,B 0,C 180,E1 -11037.078,E2 -11037.078} C_VEL
LIN {X 0,Y 416.167,Z 549.907,A -85,B 0,C 180,E1 -11037.832,E2 -11037.832} C_VEL
LIN {X 0,Y 415.151,Z 563.892,A -85,B 0,C 180,E1 -11038.773,E2 -11038.773} C_VEL
LIN {X 0,Y 414.023,Z 576.527,A -85,B 0,C 180,E1 -11039.831,E2 -11039.831} C_VEL
LIN {X 0,Y 412.648,Z 589.084,A -85,B 0,C 180,E1 -11041.102,E2 -11041.102} C_VEL
LIN {X 0,Y 411.304,Z 600.66,A -85,B 0,C 180,E1 -11042.527,E2 -11042.527} C_VEL
LIN {X 0,Y 409.947,Z 611.172,A -85,B 0,C 180,E1 -11044.078,E2 -11044.078} C_VEL
LIN {X 0,Y 408.623,Z 620.492,A -85,B 0,C 180,E1 -11045.722,E2 -11045.722} C_VEL
LIN {X 0,Y 407.558,Z 628.562,A -85,B 0,C 180,E1 -11047.439,E2 -11047.439} C_VEL
LIN {X 0,Y 406.527,Z 635.945,A -85,B 0,C 180,E1 -11049.343,E2 -11049.343} C_VEL
LIN {X 0,Y 405.698,Z 642.072,A -85,B 0,C 180,E1 -11051.309,E2 -11051.309} C_VEL
LIN {X 0,Y 405.013,Z 647.044,A -85,B 0,C 180,E1 -11053.363,E2 -11053.363} C_VEL
LIN {X 0,Y 404.637,Z 649.879,A -85,B 0,C 180,E1 -11054.899,E2 -11054.899} C_VEL
LIN {X 0,Y 404.285,Z 652.569,A -85,B 0,C 180,E1 -11056.94,E2 -11056.94} C_VEL
LIN {X 0,Y 404.092,Z 654.091,A -85,B 0,C 180,E1 -11058.971,E2 -11058.971} C_VEL
LIN {X 0,Y 404.061,Z 654.49,A -85,B 0,C 180,E1 -11060.994,E2 -11060.994} C_VEL
LIN {X 0,Y 404.131,Z 653.784,A -85,B 0,C 180,E1 -11063.008,E2 -11063.008} C_VEL
LIN {X 0,Y 404.163,Z 651.95,A -85,B 0,C 180,E1 -11065.013,E2 -11065.013} C_VEL
LIN {X 0,Y 404.192,Z 650.978,A -85,B 0,C 180,E1 -11065.74,E2 -11065.74} C_VEL
LIN {X 0,Y 403.616,Z 649.894,A -85,B 0,C 180,E1 -11066.56,E2 -11066.56} C_VEL
LIN {X 0,Y 400.97,Z 647.943,A -85,B 0,C 180,E1 -11067.896,E2 -11067.896} C_VEL
LIN {X 0,Y 398.805,Z 646.019,A -85,B 0,C 180,E1 -11068.959,E2 -11068.959} C_VEL
LIN {X 0,Y 398.008,Z 644.206,A -85,B 0,C 180,E1 -11069.762,E2 -11069.762} C_VEL
LIN {X 0,Y 398.015,Z 643.496,A -85,B 0,C 180,E1 -11070.028,E2 -11070.028} C_VEL
LIN {X 0,Y 398.791,Z 637.476,A -85,B 0,C 180,E1 -11072.02,E2 -11072.02} C_VEL
LIN {X 0,Y 399.664,Z 629.869,A -85,B 0,C 180,E1 -11074.034,E2 -11074.034} C_VEL
LIN {X 0,Y 400.61,Z 621.775,A -85,B 0,C 180,E1 -11075.79,E2 -11075.79} C_VEL
LIN {X 0,Y 401.802,Z 612.023,A -85,B 0,C 180,E1 -11077.538,E2 -11077.538} C_VEL
LIN {X 0,Y 402.868,Z 602.108,A -85,B 0,C 180,E1 -11079.033,E2 -11079.033} C_VEL
LIN {X 0,Y 403.995,Z 590.261,A -85,B 0,C 180,E1 -11080.525,E2 -11080.525} C_VEL
LIN {X 0,Y 405.277,Z 577.032,A -85,B 0,C 180,E1 -11081.884,E2 -11081.884} C_VEL
LIN {X 0,Y 406.416,Z 563.794,A -85,B 0,C 180,E1 -11082.991,E2 -11082.991} C_VEL
LIN {X 0,Y 407.369,Z 550.091,A -85,B 0,C 180,E1 -11083.913,E2 -11083.913} C_VEL
LIN {X 0,Y 408.096,Z 536.029,A -85,B 0,C 180,E1 -11084.652,E2 -11084.652} C_VEL
LIN {X 0,Y 408.568,Z 520.635,A -85,B 0,C 180,E1 -11085.248,E2 -11085.248} C_VEL
LIN {X 0,Y 408.743,Z 505.261,A -85,B 0,C 180,E1 -11085.637,E2 -11085.637} C_VEL
LIN {X 0,Y 410.282,Z 410.506,A -85,B 0,C 180,E1 -11087.329,E2 -11087.329} C_VEL
LIN {X 0,Y 400.523,Z 389.451,A -85,B 0,C 180,E1 -11088.382,E2 -11088.382} C_VEL
LIN {X 0,Y 397.295,Z 382.613,A -85,B 0,C 180,E1 -11088.74,E2 -11088.74} C_VEL
LIN {X 0,Y 397.111,Z 381.645,A -85,B 0,C 180,E1 -11088.777,E2 -11088.777} C_VEL
LIN {X 0,Y 397.091,Z 381.646,A -85,B 0,C 180,E1 -11091.819,E2 -11091.819} C_VEL
LIN {X 0,Y 397.101,Z 381.647,A -85,B 0,C 180,E1 -11095.135,E2 -11095.135} C_VEL
LIN {X 0,Y 397.06,Z 381.652,A -85,B 0,C 180,E1 -11098.548,E2 -11098.548} C_VEL
LIN {X 0,Y 397.074,Z 381.648,A -85,B 0,C 180,E1 -11101.834,E2 -11101.834} C_VEL
LIN {X 0,Y 397.114,Z 381.64,A -85,B 0,C 180,E1 -11104.494,E2 -11104.494} C_VEL
LIN {X 0,Y 397.087,Z 381.645,A -85,B 0,C 180,E1 -11108.276,E2 -11108.276} C_VEL
LIN {X 0,Y 397.043,Z 381.649,A -85,B 0,C 180,E1 -11110.914,E2 -11110.914} C_VEL
LIN {X 0,Y 397.073,Z 381.647,A -85,B 0,C 180,E1 -11114.929,E2 -11114.929} C_VEL
LIN {X 0,Y 397.047,Z 381.647,A -85,B 0,C 180,E1 -11118.023,E2 -11118.023} C_VEL
LIN {X 0,Y 397.085,Z 381.643,A -85,B 0,C 180,E1 -11121.723,E2 -11121.723} C_VEL
LIN {X 0,Y 397.111,Z 381.639,A -85,B 0,C 180,E1 -11125.505,E2 -11125.505} C_VEL
LIN {X 0,Y 397.065,Z 381.653,A -85,B 0,C 180,E1 -11129.116,E2 -11129.116} C_VEL
LIN {X 0,Y 397.051,Z 381.648,A -85,B 0,C 180,E1 -11132.252,E2 -11132.252} C_VEL
LIN {X 0,Y 397.095,Z 381.645,A -85,B 0,C 180,E1 -11134.864,E2 -11134.864} C_VEL
LIN {X 0,Y 397.088,Z 381.645,A -85,B 0,C 180,E1 -11138.181,E2 -11138.181} C_VEL
LIN {X 0,Y 397.15,Z 381.634,A -85,B 0,C 180,E1 -11141.426,E2 -11141.426} C_VEL
LIN {X 0,Y 397.165,Z 381.634,A -85,B 0,C 180,E1 -11144.607,E2 -11144.607} C_VEL
LIN {X 0,Y 397.209,Z 381.606,A -85,B 0,C 180,E1 -11147.741,E2 -11147.741} C_VEL
LIN {X 0,Y 397.219,Z 381.606,A -85,B 0,C 180,E1 -11150.837,E2 -11150.837} C_VEL
LIN {X 0,Y 397.31,Z 381.619,A -85,B 0,C 180,E1 -11153.907,E2 -11153.907} C_VEL
LIN {X 0,Y 397.424,Z 381.595,A -85,B 0,C 180,E1 -11157.973,E2 -11157.973} C_VEL
LIN {X 0,Y 397.433,Z 381.599,A -85,B 0,C 180,E1 -11162.027,E2 -11162.027} C_VEL
LIN {X 0,Y 397.304,Z 381.618,A -85,B 0,C 180,E1 -11166.092,E2 -11166.092} C_VEL
LIN {X 0,Y 397.22,Z 381.623,A -85,B 0,C 180,E1 -11169.162,E2 -11169.162} C_VEL
LIN {X 0,Y 397.209,Z 381.629,A -85,B 0,C 180,E1 -11172.258,E2 -11172.258} C_VEL
LIN {X 0,Y 397.11,Z 381.64,A -85,B 0,C 180,E1 -11175.395,E2 -11175.395} C_VEL
LIN {X 0,Y 397.079,Z 381.64,A -85,B 0,C 180,E1 -11178.577,E2 -11178.577} C_VEL
LIN {X 0,Y 397.081,Z 381.647,A -85,B 0,C 180,E1 -11181.819,E2 -11181.819} C_VEL
LIN {X 0,Y 397.095,Z 381.645,A -85,B 0,C 180,E1 -11185.136,E2 -11185.136} C_VEL
LIN {X 0,Y 397.055,Z 381.648,A -85,B 0,C 180,E1 -11188.549,E2 -11188.549} C_VEL
LIN {X 0,Y 397.072,Z 381.649,A -85,B 0,C 180,E1 -11191.836,E2 -11191.836} C_VEL
LIN {X 0,Y 397.109,Z 381.638,A -85,B 0,C 180,E1 -11194.495,E2 -11194.495} C_VEL
LIN {X 0,Y 397.082,Z 381.638,A -85,B 0,C 180,E1 -11198.277,E2 -11198.277} C_VEL
LIN {X 0,Y 397.045,Z 381.646,A -85,B 0,C 180,E1 -11201.977,E2 -11201.977} C_VEL
LIN {X 0,Y 397.079,Z 381.645,A -85,B 0,C 180,E1 -11205.07,E2 -11205.07} C_VEL
LIN {X 0,Y 397.045,Z 381.644,A -85,B 0,C 180,E1 -11208.024,E2 -11208.024} C_VEL
LIN {X 0,Y 397.097,Z 381.741,A -85,B 0,C 180,E1 -11211.607,E2 -11211.607} C_VEL
LIN {X 0,Y 402.378,Z 400.836,A -85,B 0,C 180,E1 -11214.804,E2 -11214.804} C_VEL
LIN {X 0,Y 405.707,Z 414.458,A -85,B 0,C 180,E1 -11216.949,E2 -11216.949} C_VEL
LIN {X 0,Y 404.458,Z 430.951,A -85,B 0,C 180,E1 -11219.163,E2 -11219.163} C_VEL
LIN {X 0,Y 402.854,Z 451.681,A -85,B 0,C 180,E1 -11221.92,E2 -11221.92} C_VEL
LIN {X 0,Y 409.542,Z 501.045,A -85,B 0,C 180,E1 -11223.275,E2 -11223.275} C_VEL
LIN {X 0,Y 407.424,Z 619.119,A -85,B 0,C 180,E1 -11225.374,E2 -11225.374} C_VEL
LIN {X 0,Y 406.717,Z 634.475,A -85,B 0,C 180,E1 -11225.805,E2 -11225.805} C_VEL
LIN {X 0,Y 405.59,Z 650.115,A -85,B 0,C 180,E1 -11226.446,E2 -11226.446} C_VEL
LIN {X 0,Y 404.247,Z 665.064,A -85,B 0,C 180,E1 -11227.274,E2 -11227.274} C_VEL
LIN {X 0,Y 402.953,Z 678.719,A -85,B 0,C 180,E1 -11228.246,E2 -11228.246} C_VEL
LIN {X 0,Y 401.59,Z 691.684,A -85,B 0,C 180,E1 -11229.378,E2 -11229.378} C_VEL
LIN {X 0,Y 400.369,Z 703.745,A -85,B 0,C 180,E1 -11230.651,E2 -11230.651} C_VEL
LIN {X 0,Y 399.059,Z 716.253,A -85,B 0,C 180,E1 -11232.235,E2 -11232.235} C_VEL
LIN {X 0,Y 398.057,Z 726.896,A -85,B 0,C 180,E1 -11233.854,E2 -11233.854} C_VEL
LIN {X 0,Y 397.238,Z 736.816,A -85,B 0,C 180,E1 -11235.659,E2 -11235.659} C_VEL
LIN {X 0,Y 396.663,Z 744.959,A -85,B 0,C 180,E1 -11237.432,E2 -11237.432} C_VEL
LIN {X 0,Y 396.458,Z 752.004,A -85,B 0,C 180,E1 -11239.273,E2 -11239.273} C_VEL
LIN {X 0,Y 396.347,Z 758.35,A -85,B 0,C 180,E1 -11241.331,E2 -11241.331} C_VEL
LIN {X 0,Y 396.43,Z 762.635,A -85,B 0,C 180,E1 -11243.109,E2 -11243.109} C_VEL
LIN {X 0,Y 396.52,Z 765.976,A -85,B 0,C 180,E1 -11244.915,E2 -11244.915} C_VEL
LIN {X 0,Y 396.583,Z 768.541,A -85,B 0,C 180,E1 -11246.952,E2 -11246.952} C_VEL
LIN {X 0,Y 396.822,Z 769.873,A -85,B 0,C 180,E1 -11248.985,E2 -11248.985} C_VEL
LIN {X 0,Y 396.821,Z 769.922,A -85,B 0,C 180,E1 -11251.014,E2 -11251.014} C_VEL
LIN {X 0,Y 396.565,Z 768.741,A -85,B 0,C 180,E1 -11253.047,E2 -11253.047} C_VEL
LIN {X 0,Y 396.525,Z 766.385,A -85,B 0,C 180,E1 -11255.084,E2 -11255.084} C_VEL
LIN {X 0,Y 396.368,Z 762.766,A -85,B 0,C 180,E1 -11257.129,E2 -11257.129} C_VEL
LIN {X 0,Y 396.279,Z 757.815,A -85,B 0,C 180,E1 -11259.184,E2 -11259.184} C_VEL
LIN {X 0,Y 396.447,Z 751.431,A -85,B 0,C 180,E1 -11261.244,E2 -11261.244} C_VEL
LIN {X 0,Y 396.875,Z 743.498,A -85,B 0,C 180,E1 -11263.309,E2 -11263.309} C_VEL
LIN {X 0,Y 397.546,Z 735.079,A -85,B 0,C 180,E1 -11265.114,E2 -11265.114} C_VEL
LIN {X 0,Y 398.572,Z 725.072,A -85,B 0,C 180,E1 -11266.914,E2 -11266.914} C_VEL
LIN {X 0,Y 399.73,Z 714.926,A -85,B 0,C 180,E1 -11268.449,E2 -11268.449} C_VEL
LIN {X 0,Y 401.145,Z 702.957,A -85,B 0,C 180,E1 -11269.976,E2 -11269.976} C_VEL
LIN {X 0,Y 402.729,Z 689.829,A -85,B 0,C 180,E1 -11271.363,E2 -11271.363} C_VEL
LIN {X 0,Y 404.475,Z 675.797,A -85,B 0,C 180,E1 -11272.567,E2 -11272.567} C_VEL
LIN {X 0,Y 405.884,Z 662.87,A -85,B 0,C 180,E1 -11273.468,E2 -11273.468} C_VEL
LIN {X 0,Y 407.369,Z 648.499,A -85,B 0,C 180,E1 -11274.255,E2 -11274.255} C_VEL
LIN {X 0,Y 408.658,Z 632.99,A -85,B 0,C 180,E1 -11274.884,E2 -11274.884} C_VEL
LIN {X 0,Y 409.543,Z 617.835,A -85,B 0,C 180,E1 -11275.302,E2 -11275.302} C_VEL
LIN {X 0,Y 411.97,Z 501.899,A -85,B 0,C 180,E1 -11277.399,E2 -11277.399} C_VEL
LIN {X 0,Y 408.335,Z 473.994,A -85,B 0,C 180,E1 -11278.238,E2 -11278.238} C_VEL
LIN {X 0,Y 404.349,Z 449.828,A -85,B 0,C 180,E1 -11279.082,E2 -11279.082} C_VEL
LIN {X 0,Y 406.895,Z 423.823,A -85,B 0,C 180,E1 -11282.666,E2 -11282.666} C_VEL
LIN {X 0,Y 407.398,Z 417.869,A -85,B 0,C 180,E1 -11283.505,E2 -11283.505} C_VEL
LIN {X 0,Y 404.345,Z 405.292,A -85,B 0,C 180,E1 -11285.653,E2 -11285.653} C_VEL
LIN {X 0,Y 399.361,Z 388.923,A -85,B 0,C 180,E1 -11288.695,E2 -11288.695} C_VEL
LIN {X 0,Y 397.084,Z 381.649,A -85,B 0,C 180,E1 -11290.145,E2 -11290.145} C_VEL
LIN {X 0,Y 397.088,Z 381.647,A -85,B 0,C 180,E1 -11293.648,E2 -11293.648} C_VEL
LIN {X 0,Y 397.081,Z 381.636,A -85,B 0,C 180,E1 -11296.522,E2 -11296.522} C_VEL
LIN {X 0,Y 397.075,Z 381.647,A -85,B 0,C 180,E1 -11300.419,E2 -11300.419} C_VEL
LIN {X 0,Y 397.082,Z 381.646,A -85,B 0,C 180,E1 -11303.003,E2 -11303.003} C_VEL
LIN {X 0,Y 397.1,Z 381.643,A -85,B 0,C 180,E1 -11306.726,E2 -11306.726} C_VEL
LIN {X 0,Y 397.104,Z 381.646,A -85,B 0,C 180,E1 -11310.294,E2 -11310.294} C_VEL
LIN {X 0,Y 397.062,Z 381.65,A -85,B 0,C 180,E1 -11313.737,E2 -11313.737} C_VEL
LIN {X 0,Y 397.087,Z 381.648,A -85,B 0,C 180,E1 -11317.085,E2 -11317.085} C_VEL
LIN {X 0,Y 397.082,Z 381.65,A -85,B 0,C 180,E1 -11320.35,E2 -11320.35} C_VEL
LIN {X 0,Y 397.106,Z 381.642,A -85,B 0,C 180,E1 -11323.551,E2 -11323.551} C_VEL
LIN {X 0,Y 397.217,Z 381.63,A -85,B 0,C 180,E1 -11326.703,E2 -11326.703} C_VEL
LIN {X 0,Y 397.195,Z 381.628,A -85,B 0,C 180,E1 -11329.809,E2 -11329.809} C_VEL
LIN {X 0,Y 397.275,Z 381.618,A -85,B 0,C 180,E1 -11332.887,E2 -11332.887} C_VEL
LIN {X 0,Y 397.214,Z 381.632,A -85,B 0,C 180,E1 -11334.925,E2 -11334.925} C_VEL
LIN {X 0,Y 397.429,Z 381.597,A -85,B 0,C 180,E1 -11337.973,E2 -11337.973} C_VEL
LIN {X 0,Y 397.426,Z 381.599,A -85,B 0,C 180,E1 -11342.027,E2 -11342.027} C_VEL
LIN {X 0,Y 397.308,Z 381.593,A -85,B 0,C 180,E1 -11346.709,E2 -11346.709} C_VEL
LIN {X 0,Y 397.198,Z 381.63,A -85,B 0,C 180,E1 -11350.192,E2 -11350.192} C_VEL
LIN {X 0,Y 397.215,Z 381.613,A -85,B 0,C 180,E1 -11353.322,E2 -11353.322} C_VEL
LIN {X 0,Y 397.171,Z 381.637,A -85,B 0,C 180,E1 -11357.156,E2 -11357.156} C_VEL
LIN {X 0,Y 397.091,Z 381.628,A -85,B 0,C 180,E1 -11360.731,E2 -11360.731} C_VEL
LIN {X 0,Y 397.096,Z 381.645,A -85,B 0,C 180,E1 -11364.021,E2 -11364.021} C_VEL
LIN {X 0,Y 397.057,Z 381.639,A -85,B 0,C 180,E1 -11367.401,E2 -11367.401} C_VEL
LIN {X 0,Y 397.089,Z 381.647,A -85,B 0,C 180,E1 -11369.864,E2 -11369.864} C_VEL
LIN {X 0,Y 397.103,Z 381.643,A -85,B 0,C 180,E1 -11373.274,E2 -11373.274} C_VEL
LIN {X 0,Y 397.089,Z 381.639,A -85,B 0,C 180,E1 -11376.996,E2 -11376.996} C_VEL
LIN {X 0,Y 397.048,Z 381.645,A -85,B 0,C 180,E1 -11380.439,E2 -11380.439} C_VEL
LIN {X 0,Y 397.081,Z 381.639,A -85,B 0,C 180,E1 -11383.652,E2 -11383.652} C_VEL
LIN {X 0,Y 397.092,Z 381.643,A -85,B 0,C 180,E1 -11386.523,E2 -11386.523} C_VEL
LIN {X 0,Y 397.082,Z 381.646,A -85,B 0,C 180,E1 -11390.421,E2 -11390.421} C_VEL
LIN {X 0,Y 397.087,Z 381.642,A -85,B 0,C 180,E1 -11391.889,E2 -11391.889} C_VEL
LIN {X 0,Y 398.117,Z 384.523,A -85,B 0,C 180,E1 -11392.057,E2 -11392.057} C_VEL
LIN {X 0,Y 399.608,Z 386.989,A -85,B 0,C 180,E1 -11392.248,E2 -11392.248} C_VEL
LIN {X 0,Y 409.225,Z 404.367,A -85,B 0,C 180,E1 -11393.458,E2 -11393.458} C_VEL
LIN {X 0,Y 413.449,Z 412.891,A -85,B 0,C 180,E1 -11393.983,E2 -11393.983} C_VEL
LIN {X 0,Y 411.513,Z 507.471,A -85,B 0,C 180,E1 -11395.697,E2 -11395.697} C_VEL
LIN {X 0,Y 411.257,Z 523.107,A -85,B 0,C 180,E1 -11396.116,E2 -11396.116} C_VEL
LIN {X 0,Y 410.721,Z 536.777,A -85,B 0,C 180,E1 -11396.655,E2 -11396.655} C_VEL
LIN {X 0,Y 409.838,Z 551.136,A -85,B 0,C 180,E1 -11397.415,E2 -11397.415} C_VEL
LIN {X 0,Y 408.783,Z 565.122,A -85,B 0,C 180,E1 -11398.375,E2 -11398.375} C_VEL
LIN {X 0,Y 407.578,Z 578.053,A -85,B 0,C 180,E1 -11399.479,E2 -11399.479} C_VEL
LIN {X 0,Y 406.169,Z 590.24,A -85,B 0,C 180,E1 -11400.739,E2 -11400.739} C_VEL
LIN {X 0,Y 404.725,Z 601.984,A -85,B 0,C 180,E1 -11402.21,E2 -11402.21} C_VEL
LIN {X 0,Y 403.419,Z 611.468,A -85,B 0,C 180,E1 -11403.627,E2 -11403.627} C_VEL
LIN {X 0,Y 401.962,Z 621.4,A -85,B 0,C 180,E1 -11405.393,E2 -11405.393} C_VEL
LIN {X 0,Y 400.709,Z 630.192,A -85,B 0,C 180,E1 -11407.304,E2 -11407.304} C_VEL
LIN {X 0,Y 399.813,Z 636.17,A -85,B 0,C 180,E1 -11408.858,E2 -11408.858} C_VEL
LIN {X 0,Y 398.87,Z 642.779,A -85,B 0,C 180,E1 -11410.977,E2 -11410.977} C_VEL
LIN {X 0,Y 398.135,Z 647.831,A -85,B 0,C 180,E1 -11413.067,E2 -11413.067} C_VEL
LIN {X 0,Y 397.703,Z 650.705,A -85,B 0,C 180,E1 -11414.63,E2 -11414.63} C_VEL
LIN {X 0,Y 397.317,Z 653.467,A -85,B 0,C 180,E1 -11416.706,E2 -11416.706} C_VEL
LIN {X 0,Y 397.089,Z 655.06,A -85,B 0,C 180,E1 -11418.774,E2 -11418.774} C_VEL
LIN {X 0,Y 397.041,Z 655.529,A -85,B 0,C 180,E1 -11420.834,E2 -11420.834} C_VEL
LIN {X 0,Y 397.105,Z 654.857,A -85,B 0,C 180,E1 -11422.884,E2 -11422.884} C_VEL
LIN {X 0,Y 397.141,Z 653.088,A -85,B 0,C 180,E1 -11424.924,E2 -11424.924} C_VEL
LIN {X 0,Y 397.454,Z 650.169,A -85,B 0,C 180,E1 -11426.96,E2 -11426.96} C_VEL
LIN {X 0,Y 397.755,Z 646.09,A -85,B 0,C 180,E1 -11428.988,E2 -11428.988} C_VEL
LIN {X 0,Y 398.015,Z 643.496,A -85,B 0,C 180,E1 -11430.028,E2 -11430.028} C_VEL
LIN {X 0,Y 397.653,Z 641.42,A -85,B 0,C 180,E1 -11430.821,E2 -11430.821} C_VEL
LIN {X 0,Y 395.367,Z 637.919,A -85,B 0,C 180,E1 -11432.123,E2 -11432.123} C_VEL
LIN {X 0,Y 393.091,Z 633.978,A -85,B 0,C 180,E1 -11433.407,E2 -11433.407} C_VEL
LIN {X 0,Y 392.746,Z 631.118,A -85,B 0,C 180,E1 -11434.162,E2 -11434.162} C_VEL
LIN {X 0,Y 393.678,Z 623.366,A -85,B 0,C 180,E1 -11435.892,E2 -11435.892} C_VEL
LIN {X 0,Y 394.926,Z 613.726,A -85,B 0,C 180,E1 -11437.67,E2 -11437.67} C_VEL
LIN {X 0,Y 396.021,Z 603.894,A -85,B 0,C 180,E1 -11439.191,E2 -11439.191} C_VEL
LIN {X 0,Y 397.221,Z 592.199,A -85,B 0,C 180,E1 -11440.706,E2 -11440.706} C_VEL
LIN {X 0,Y 398.481,Z 579.234,A -85,B 0,C 180,E1 -11442.09,E2 -11442.09} C_VEL
LIN {X 0,Y 399.683,Z 566.227,A -85,B 0,C 180,E1 -11443.214,E2 -11443.214} C_VEL
LIN {X 0,Y 400.723,Z 551.88,A -85,B 0,C 180,E1 -11444.214,E2 -11444.214} C_VEL
LIN {X 0,Y 401.545,Z 536.733,A -85,B 0,C 180,E1 -11445.026,E2 -11445.026} C_VEL
LIN {X 0,Y 402.037,Z 521.052,A -85,B 0,C 180,E1 -11445.636,E2 -11445.636} C_VEL
LIN {X 0,Y 402.212,Z 505.759,A -85,B 0,C 180,E1 -11446.023,E2 -11446.023} C_VEL
LIN {X 0,Y 403.763,Z 412.22,A -85,B 0,C 180,E1 -11447.721,E2 -11447.721} C_VEL
LIN {X 0,Y 393.78,Z 390.923,A -85,B 0,C 180,E1 -11448.823,E2 -11448.823} C_VEL
LIN {X 0,Y 390.244,Z 383.38,A -85,B 0,C 180,E1 -11449.229,E2 -11449.229} C_VEL
LIN {X 0,Y 390.078,Z 382.521,A -85,B 0,C 180,E1 -11449.264,E2 -11449.264} C_VEL
LIN {X 0,Y 390.033,Z 382.525,A -85,B 0,C 180,E1 -11452.234,E2 -11452.234} C_VEL
LIN {X 0,Y 390.051,Z 382.525,A -85,B 0,C 180,E1 -11455.722,E2 -11455.722} C_VEL
LIN {X 0,Y 390.021,Z 382.518,A -85,B 0,C 180,E1 -11459.112,E2 -11459.112} C_VEL
LIN {X 0,Y 390.038,Z 382.527,A -85,B 0,C 180,E1 -11462.721,E2 -11462.721} C_VEL
LIN {X 0,Y 390.04,Z 382.523,A -85,B 0,C 180,E1 -11465.821,E2 -11465.821} C_VEL
LIN {X 0,Y 390.034,Z 382.524,A -85,B 0,C 180,E1 -11469.211,E2 -11469.211} C_VEL
LIN {X 0,Y 390.004,Z 382.527,A -85,B 0,C 180,E1 -11472.367,E2 -11472.367} C_VEL
LIN {X 0,Y 390.039,Z 382.522,A -85,B 0,C 180,E1 -11476.115,E2 -11476.115} C_VEL
LIN {X 0,Y 390.006,Z 382.531,A -85,B 0,C 180,E1 -11479.554,E2 -11479.554} C_VEL
LIN {X 0,Y 390.033,Z 382.52,A -85,B 0,C 180,E1 -11482.45,E2 -11482.45} C_VEL
LIN {X 0,Y 390.057,Z 382.514,A -85,B 0,C 180,E1 -11486.044,E2 -11486.044} C_VEL
LIN {X 0,Y 390.035,Z 382.521,A -85,B 0,C 180,E1 -11489.87,E2 -11489.87} C_VEL
LIN {X 0,Y 390.019,Z 382.53,A -85,B 0,C 180,E1 -11493.225,E2 -11493.225} C_VEL
LIN {X 0,Y 390.053,Z 382.516,A -85,B 0,C 180,E1 -11496.766,E2 -11496.766} C_VEL
LIN {X 0,Y 390.097,Z 382.512,A -85,B 0,C 180,E1 -11499.982,E2 -11499.982} C_VEL
LIN {X 0,Y 390.13,Z 382.513,A -85,B 0,C 180,E1 -11503.248,E2 -11503.248} C_VEL
LIN {X 0,Y 390.189,Z 382.495,A -85,B 0,C 180,E1 -11506.561,E2 -11506.561} C_VEL
LIN {X 0,Y 390.151,Z 382.477,A -85,B 0,C 180,E1 -11509.622,E2 -11509.622} C_VEL
LIN {X 0,Y 390.237,Z 382.492,A -85,B 0,C 180,E1 -11512.757,E2 -11512.757} C_VEL
LIN {X 0,Y 390.187,Z 382.504,A -85,B 0,C 180,E1 -11514.833,E2 -11514.833} C_VEL
LIN {X 0,Y 390.391,Z 382.471,A -85,B 0,C 180,E1 -11517.936,E2 -11517.936} C_VEL
LIN {X 0,Y 390.4,Z 382.475,A -85,B 0,C 180,E1 -11522.063,E2 -11522.063} C_VEL
LIN {X 0,Y 390.259,Z 382.495,A -85,B 0,C 180,E1 -11526.203,E2 -11526.203} C_VEL
LIN {X 0,Y 390.179,Z 382.5,A -85,B 0,C 180,E1 -11529.329,E2 -11529.329} C_VEL
LIN {X 0,Y 390.161,Z 382.506,A -85,B 0,C 180,E1 -11532.483,E2 -11532.483} C_VEL
LIN {X 0,Y 390.053,Z 382.523,A -85,B 0,C 180,E1 -11535.68,E2 -11535.68} C_VEL
LIN {X 0,Y 390.035,Z 382.518,A -85,B 0,C 180,E1 -11538.925,E2 -11538.925} C_VEL
LIN {X 0,Y 390.023,Z 382.522,A -85,B 0,C 180,E1 -11542.235,E2 -11542.235} C_VEL
LIN {X 0,Y 390.043,Z 382.524,A -85,B 0,C 180,E1 -11545.722,E2 -11545.722} C_VEL
LIN {X 0,Y 390.016,Z 382.526,A -85,B 0,C 180,E1 -11549.113,E2 -11549.113} C_VEL
LIN {X 0,Y 390.034,Z 382.519,A -85,B 0,C 180,E1 -11552.722,E2 -11552.722} C_VEL
LIN {X 0,Y 390.035,Z 382.528,A -85,B 0,C 180,E1 -11555.822,E2 -11555.822} C_VEL
LIN {X 0,Y 390.029,Z 382.518,A -85,B 0,C 180,E1 -11559.212,E2 -11559.212} C_VEL
LIN {X 0,Y 390.024,Z 382.519,A -85,B 0,C 180,E1 -11562.372,E2 -11562.372} C_VEL
LIN {X 0,Y 390.035,Z 382.521,A -85,B 0,C 180,E1 -11565.354,E2 -11565.354} C_VEL
LIN {X 0,Y 390.009,Z 382.518,A -85,B 0,C 180,E1 -11568.185,E2 -11568.185} C_VEL
LIN {X 0,Y 390.051,Z 382.527,A -85,B 0,C 180,E1 -11571.154,E2 -11571.154} C_VEL
LIN {X 0,Y 395.004,Z 400.361,A -85,B 0,C 180,E1 -11574.221,E2 -11574.221} C_VEL
LIN {X 0,Y 398.749,Z 415.598,A -85,B 0,C 180,E1 -11576.678,E2 -11576.678} C_VEL
LIN {X 0,Y 398.881,Z 418.099,A -85,B 0,C 180,E1 -11577.042,E2 -11577.042} C_VEL
LIN {X 0,Y 396.434,Z 447.022,A -85,B 0,C 180,E1 -11580.968,E2 -11580.968} C_VEL
LIN {X 0,Y 396.101,Z 450.6,A -85,B 0,C 180,E1 -11581.449,E2 -11581.449} C_VEL
LIN {X 0,Y 403.03,Z 502.131,A -85,B 0,C 180,E1 -11582.9,E2 -11582.9} C_VEL
LIN {X 0,Y 400.825,Z 618.956,A -85,B 0,C 180,E1 -11585.011,E2 -11585.011} C_VEL
LIN {X 0,Y 400.031,Z 634.912,A -85,B 0,C 180,E1 -11585.477,E2 -11585.477} C_VEL
LIN {X 0,Y 398.824,Z 650.628,A -85,B 0,C 180,E1 -11586.15,E2 -11586.15} C_VEL
LIN {X 0,Y 397.45,Z 665.231,A -85,B 0,C 180,E1 -11586.993,E2 -11586.993} C_VEL
LIN {X 0,Y 395.958,Z 680.333,A -85,B 0,C 180,E1 -11588.116,E2 -11588.116} C_VEL
LIN {X 0,Y 394.583,Z 692.854,A -85,B 0,C 180,E1 -11589.268,E2 -11589.268} C_VEL
LIN {X 0,Y 393.315,Z 704.545,A -85,B 0,C 180,E1 -11590.561,E2 -11590.561} C_VEL
LIN {X 0,Y 392.054,Z 715.994,A -85,B 0,C 180,E1 -11592.065,E2 -11592.065} C_VEL
LIN {X 0,Y 390.953,Z 727.152,A -85,B 0,C 180,E1 -11593.821,E2 -11593.821} C_VEL
LIN {X 0,Y 390.142,Z 736.862,A -85,B 0,C 180,E1 -11595.659,E2 -11595.659} C_VEL
LIN {X 0,Y 389.583,Z 744.954,A -85,B 0,C 180,E1 -11597.498,E2 -11597.498} C_VEL
LIN {X 0,Y 389.327,Z 752.54,A -85,B 0,C 180,E1 -11599.6,E2 -11599.6} C_VEL
LIN {X 0,Y 389.31,Z 758.546,A -85,B 0,C 180,E1 -11601.696,E2 -11601.696} C_VEL
LIN {X 0,Y 389.364,Z 763.112,A -85,B 0,C 180,E1 -11603.782,E2 -11603.782} C_VEL
LIN {X 0,Y 389.541,Z 766.361,A -85,B 0,C 180,E1 -11605.861,E2 -11605.861} C_VEL
LIN {X 0,Y 389.575,Z 768.317,A -85,B 0,C 180,E1 -11607.932,E2 -11607.932} C_VEL
LIN {X 0,Y 389.796,Z 768.84,A -85,B 0,C 180,E1 -11608.967,E2 -11608.967} C_VEL
LIN {X 0,Y 389.794,Z 768.911,A -85,B 0,C 180,E1 -11611.033,E2 -11611.033} C_VEL
LIN {X 0,Y 389.524,Z 767.749,A -85,B 0,C 180,E1 -11613.102,E2 -11613.102} C_VEL
LIN {X 0,Y 389.456,Z 765.41,A -85,B 0,C 180,E1 -11615.176,E2 -11615.176} C_VEL
LIN {X 0,Y 389.297,Z 761.813,A -85,B 0,C 180,E1 -11617.259,E2 -11617.259} C_VEL
LIN {X 0,Y 389.215,Z 756.874,A -85,B 0,C 180,E1 -11619.352,E2 -11619.352} C_VEL
LIN {X 0,Y 389.39,Z 750.513,A -85,B 0,C 180,E1 -11621.451,E2 -11621.451} C_VEL
LIN {X 0,Y 389.849,Z 742.611,A -85,B 0,C 180,E1 -11623.553,E2 -11623.553} C_VEL
LIN {X 0,Y 390.675,Z 732.948,A -85,B 0,C 180,E1 -11625.654,E2 -11625.654} C_VEL
LIN {X 0,Y 391.846,Z 722.74,A -85,B 0,C 180,E1 -11627.482,E2 -11627.482} C_VEL
LIN {X 0,Y 393.13,Z 712.359,A -85,B 0,C 180,E1 -11629.041,E2 -11629.041} C_VEL
LIN {X 0,Y 394.627,Z 700.103,A -85,B 0,C 180,E1 -11630.592,E2 -11630.592} C_VEL
LIN {X 0,Y 396.219,Z 687.933,A -85,B 0,C 180,E1 -11631.868,E2 -11631.868} C_VEL
LIN {X 0,Y 397.988,Z 674.478,A -85,B 0,C 180,E1 -11633.028,E2 -11633.028} C_VEL
LIN {X 0,Y 399.615,Z 660.556,A -85,B 0,C 180,E1 -11633.996,E2 -11633.996} C_VEL
LIN {X 0,Y 401.163,Z 645.809,A -85,B 0,C 180,E1 -11634.793,E2 -11634.793} C_VEL
LIN {X 0,Y 402.484,Z 630.557,A -85,B 0,C 180,E1 -11635.397,E2 -11635.397} C_VEL
LIN {X 0,Y 403.291,Z 614.55,A -85,B 0,C 180,E1 -11635.827,E2 -11635.827} C_VEL
LIN {X 0,Y 405.765,Z 503.567,A -85,B 0,C 180,E1 -11637.854,E2 -11637.854} C_VEL
LIN {X 0,Y 402.856,Z 479.735,A -85,B 0,C 180,E1 -11638.571,E2 -11638.571} C_VEL
LIN {X 0,Y 397.82,Z 448.861,A -85,B 0,C 180,E1 -11639.646,E2 -11639.646} C_VEL
LIN {X 0,Y 400.485,Z 423.181,A -85,B 0,C 180,E1 -11643.256,E2 -11643.256} C_VEL
LIN {X 0,Y 400.75,Z 419.754,A -85,B 0,C 180,E1 -11643.752,E2 -11643.752} C_VEL
LIN {X 0,Y 397.571,Z 406.994,A -85,B 0,C 180,E1 -11645.987,E2 -11645.987} C_VEL
LIN {X 0,Y 392.572,Z 390.475,A -85,B 0,C 180,E1 -11649.131,E2 -11649.131} C_VEL
LIN {X 0,Y 389.997,Z 382.529,A -85,B 0,C 180,E1 -11650.776,E2 -11650.776} C_VEL
LIN {X 0,Y 390.043,Z 382.523,A -85,B 0,C 180,E1 -11653.885,E2 -11653.885} C_VEL
LIN {X 0,Y 390.037,Z 382.517,A -85,B 0,C 180,E1 -11656.787,E2 -11656.787} C_VEL
LIN {X 0,Y 390,Z 382.528,A -85,B 0,C 180,E1 -11659.554,E2 -11659.554} C_VEL
LIN {X 0,Y 390.027,Z 382.529,A -85,B 0,C 180,E1 -11662.45,E2 -11662.45} C_VEL
LIN {X 0,Y 390.051,Z 382.523,A -85,B 0,C 180,E1 -11666.044,E2 -11666.044} C_VEL
LIN {X 0,Y 390.031,Z 382.523,A -85,B 0,C 180,E1 -11669.87,E2 -11669.87} C_VEL
LIN {X 0,Y 390.018,Z 382.527,A -85,B 0,C 180,E1 -11673.225,E2 -11673.225} C_VEL
LIN {X 0,Y 390.046,Z 382.528,A -85,B 0,C 180,E1 -11676.767,E2 -11676.767} C_VEL
LIN {X 0,Y 390.057,Z 382.521,A -85,B 0,C 180,E1 -11679.981,E2 -11679.981} C_VEL
LIN {X 0,Y 390.069,Z 382.519,A -85,B 0,C 180,E1 -11683.245,E2 -11683.245} C_VEL
LIN {X 0,Y 390.159,Z 382.508,A -85,B 0,C 180,E1 -11686.576,E2 -11686.576} C_VEL
LIN {X 0,Y 390.147,Z 382.506,A -85,B 0,C 180,E1 -11689.622,E2 -11689.622} C_VEL
LIN {X 0,Y 390.229,Z 382.497,A -85,B 0,C 180,E1 -11692.758,E2 -11692.758} C_VEL
LIN {X 0,Y 390.185,Z 382.509,A -85,B 0,C 180,E1 -11694.833,E2 -11694.833} C_VEL
LIN {X 0,Y 390.396,Z 382.473,A -85,B 0,C 180,E1 -11697.937,E2 -11697.937} C_VEL
LIN {X 0,Y 390.394,Z 382.475,A -85,B 0,C 180,E1 -11702.064,E2 -11702.064} C_VEL
LIN {X 0,Y 390.261,Z 382.47,A -85,B 0,C 180,E1 -11706.705,E2 -11706.705} C_VEL
LIN {X 0,Y 390.176,Z 382.504,A -85,B 0,C 180,E1 -11709.33,E2 -11709.33} C_VEL
LIN {X 0,Y 390.157,Z 382.502,A -85,B 0,C 180,E1 -11712.484,E2 -11712.484} C_VEL
LIN {X 0,Y 390.126,Z 382.503,A -85,B 0,C 180,E1 -11715.678,E2 -11715.678} C_VEL
LIN {X 0,Y 390.091,Z 382.512,A -85,B 0,C 180,E1 -11718.923,E2 -11718.923} C_VEL
LIN {X 0,Y 390.023,Z 382.515,A -85,B 0,C 180,E1 -11722.235,E2 -11722.235} C_VEL
LIN {X 0,Y 390.04,Z 382.515,A -85,B 0,C 180,E1 -11725.723,E2 -11725.723} C_VEL
LIN {X 0,Y 390.016,Z 382.532,A -85,B 0,C 180,E1 -11729.113,E2 -11729.113} C_VEL
LIN {X 0,Y 390.032,Z 382.515,A -85,B 0,C 180,E1 -11732.723,E2 -11732.723} C_VEL
LIN {X 0,Y 390.035,Z 382.521,A -85,B 0,C 180,E1 -11735.824,E2 -11735.824} C_VEL
LIN {X 0,Y 390.031,Z 382.526,A -85,B 0,C 180,E1 -11739.214,E2 -11739.214} C_VEL
LIN {X 0,Y 390.024,Z 382.527,A -85,B 0,C 180,E1 -11742.373,E2 -11742.373} C_VEL
LIN {X 0,Y 390.037,Z 382.527,A -85,B 0,C 180,E1 -11745.355,E2 -11745.355} C_VEL
LIN {X 0,Y 390.012,Z 382.528,A -85,B 0,C 180,E1 -11748.186,E2 -11748.186} C_VEL
LIN {X 0,Y 390.052,Z 382.577,A -85,B 0,C 180,E1 -11751.243,E2 -11751.243} C_VEL
LIN {X 0,Y 391.01,Z 385.319,A -85,B 0,C 180,E1 -11751.396,E2 -11751.396} C_VEL
LIN {X 0,Y 392.626,Z 387.941,A -85,B 0,C 180,E1 -11751.609,E2 -11751.609} C_VEL
LIN {X 0,Y 401.65,Z 403.925,A -85,B 0,C 180,E1 -11752.787,E2 -11752.787} C_VEL
LIN {X 0,Y 407.254,Z 414.862,A -85,B 0,C 180,E1 -11753.502,E2 -11753.502} C_VEL
LIN {X 0,Y 405.32,Z 507.688,A -85,B 0,C 180,E1 -11755.211,E2 -11755.211} C_VEL
LIN {X 0,Y 405.081,Z 522.639,A -85,B 0,C 180,E1 -11755.603,E2 -11755.603} C_VEL
LIN {X 0,Y 404.539,Z 536.635,A -85,B 0,C 180,E1 -11756.152,E2 -11756.152} C_VEL
LIN {X 0,Y 403.603,Z 551.471,A -85,B 0,C 180,E1 -11756.934,E2 -11756.934} C_VEL
LIN {X 0,Y 402.59,Z 564.575,A -85,B 0,C 180,E1 -11757.831,E2 -11757.831} C_VEL
LIN {X 0,Y 401.371,Z 577.037,A -85,B 0,C 180,E1 -11758.878,E2 -11758.878} C_VEL
LIN {X 0,Y 399.963,Z 589.04,A -85,B 0,C 180,E1 -11760.094,E2 -11760.094} C_VEL
LIN {X 0,Y 398.454,Z 600.971,A -85,B 0,C 180,E1 -11761.562,E2 -11761.562} C_VEL
LIN {X 0,Y 396.909,Z 611.775,A -85,B 0,C 180,E1 -11763.16,E2 -11763.16} C_VEL
LIN {X 0,Y 395.564,Z 620.838,A -85,B 0,C 180,E1 -11764.761,E2 -11764.761} C_VEL
LIN {X 0,Y 394.219,Z 629.624,A -85,B 0,C 180,E1 -11766.631,E2 -11766.631} C_VEL
LIN {X 0,Y 393.009,Z 637.182,A -85,B 0,C 180,E1 -11768.593,E2 -11768.593} C_VEL
LIN {X 0,Y 392.046,Z 643.493,A -85,B 0,C 180,E1 -11770.633,E2 -11770.633} C_VEL
LIN {X 0,Y 391.258,Z 648.622,A -85,B 0,C 180,E1 -11772.76,E2 -11772.76} C_VEL
LIN {X 0,Y 390.767,Z 651.535,A -85,B 0,C 180,E1 -11774.35,E2 -11774.35} C_VEL
LIN {X 0,Y 390.333,Z 654.384,A -85,B 0,C 180,E1 -11776.479,E2 -11776.479} C_VEL
LIN {X 0,Y 390.098,Z 656.03,A -85,B 0,C 180,E1 -11778.57,E2 -11778.57} C_VEL
LIN {X 0,Y 390.035,Z 656.553,A -85,B 0,C 180,E1 -11780.668,E2 -11780.668} C_VEL
LIN {X 0,Y 390.067,Z 655.929,A -85,B 0,C 180,E1 -11782.755,E2 -11782.755} C_VEL
LIN {X 0,Y 390.118,Z 654.225,A -85,B 0,C 180,E1 -11784.833,E2 -11784.833} C_VEL
LIN {X 0,Y 390.43,Z 651.376,A -85,B 0,C 180,E1 -11786.905,E2 -11786.905} C_VEL
LIN {X 0,Y 390.753,Z 647.369,A -85,B 0,C 180,E1 -11788.97,E2 -11788.97} C_VEL
LIN {X 0,Y 391.371,Z 642.063,A -85,B 0,C 180,E1 -11791.029,E2 -11791.029} C_VEL
LIN {X 0,Y 392.252,Z 635.318,A -85,B 0,C 180,E1 -11793.082,E2 -11793.082} C_VEL
LIN {X 0,Y 392.746,Z 631.118,A -85,B 0,C 180,E1 -11794.162,E2 -11794.162} C_VEL
LIN {X 0,Y 392.432,Z 628.175,A -85,B 0,C 180,E1 -11794.903,E2 -11794.903} C_VEL
LIN {X 0,Y 388.618,Z 619.025,A -85,B 0,C 180,E1 -11797.088,E2 -11797.088} C_VEL
LIN {X 0,Y 388.097,Z 615.496,A -85,B 0,C 180,E1 -11797.783,E2 -11797.783} C_VEL
LIN {X 0,Y 388.174,Z 614.217,A -85,B 0,C 180,E1 -11798.005,E2 -11798.005} C_VEL
LIN {X 0,Y 389.378,Z 603.905,A -85,B 0,C 180,E1 -11799.611,E2 -11799.611} C_VEL
LIN {X 0,Y 390.607,Z 592.005,A -85,B 0,C 180,E1 -11801.153,E2 -11801.153} C_VEL
LIN {X 0,Y 391.837,Z 580.079,A -85,B 0,C 180,E1 -11802.429,E2 -11802.429} C_VEL
LIN {X 0,Y 393.078,Z 567.041,A -85,B 0,C 180,E1 -11803.572,E2 -11803.572} C_VEL
LIN {X 0,Y 394.164,Z 552.635,A -85,B 0,C 180,E1 -11804.587,E2 -11804.587} C_VEL
LIN {X 0,Y 395.01,Z 537.389,A -85,B 0,C 180,E1 -11805.413,E2 -11805.413} C_VEL
LIN {X 0,Y 395.505,Z 522.146,A -85,B 0,C 180,E1 -11806.014,E2 -11806.014} C_VEL
LIN {X 0,Y 395.71,Z 506.012,A -85,B 0,C 180,E1 -11806.424,E2 -11806.424} C_VEL
LIN {X 0,Y 397.346,Z 414.287,A -85,B 0,C 180,E1 -11808.112,E2 -11808.112} C_VEL
LIN {X 0,Y 386.618,Z 391.453,A -85,B 0,C 180,E1 -11809.33,E2 -11809.33} C_VEL
LIN {X 0,Y 383.253,Z 384.519,A -85,B 0,C 180,E1 -11809.722,E2 -11809.722} C_VEL
LIN {X 0,Y 383.044,Z 383.397,A -85,B 0,C 180,E1 -11809.777,E2 -11809.777} C_VEL
LIN {X 0,Y 383.005,Z 383.402,A -85,B 0,C 180,E1 -11813.809,E2 -11813.809} C_VEL
LIN {X 0,Y 382.966,Z 383.41,A -85,B 0,C 180,E1 -11817.309,E2 -11817.309} C_VEL
LIN {X 0,Y 382.978,Z 383.394,A -85,B 0,C 180,E1 -11820.919,E2 -11820.919} C_VEL
LIN {X 0,Y 383.01,Z 383.399,A -85,B 0,C 180,E1 -11824.668,E2 -11824.668} C_VEL
LIN {X 0,Y 382.99,Z 383.402,A -85,B 0,C 180,E1 -11827.901,E2 -11827.901} C_VEL
LIN {X 0,Y 382.954,Z 383.41,A -85,B 0,C 180,E1 -11831.351,E2 -11831.351} C_VEL
LIN {X 0,Y 382.961,Z 383.401,A -85,B 0,C 180,E1 -11834.297,E2 -11834.297} C_VEL
LIN {X 0,Y 382.978,Z 383.401,A -85,B 0,C 180,E1 -11837.235,E2 -11837.235} C_VEL
LIN {X 0,Y 382.981,Z 383.402,A -85,B 0,C 180,E1 -11840.418,E2 -11840.418} C_VEL
LIN {X 0,Y 383.009,Z 383.4,A -85,B 0,C 180,E1 -11844.042,E2 -11844.042} C_VEL
LIN {X 0,Y 382.976,Z 383.407,A -85,B 0,C 180,E1 -11847.579,E2 -11847.579} C_VEL
LIN {X 0,Y 382.967,Z 383.4,A -85,B 0,C 180,E1 -11850.298,E2 -11850.298} C_VEL
LIN {X 0,Y 382.997,Z 383.4,A -85,B 0,C 180,E1 -11854.045,E2 -11854.045} C_VEL
LIN {X 0,Y 382.98,Z 383.402,A -85,B 0,C 180,E1 -11857.333,E2 -11857.333} C_VEL
LIN {X 0,Y 383.051,Z 383.389,A -85,B 0,C 180,E1 -11860.716,E2 -11860.716} C_VEL
LIN {X 0,Y 383.069,Z 383.391,A -85,B 0,C 180,E1 -11864.026,E2 -11864.026} C_VEL
LIN {X 0,Y 383.128,Z 383.364,A -85,B 0,C 180,E1 -11867.283,E2 -11867.283} C_VEL
LIN {X 0,Y 383.13,Z 383.359,A -85,B 0,C 180,E1 -11870.497,E2 -11870.497} C_VEL
LIN {X 0,Y 383.224,Z 383.375,A -85,B 0,C 180,E1 -11873.682,E2 -11873.682} C_VEL
LIN {X 0,Y 383.356,Z 383.347,A -85,B 0,C 180,E1 -11877.898,E2 -11877.898} C_VEL
LIN {X 0,Y 383.366,Z 383.35,A -85,B 0,C 180,E1 -11882.101,E2 -11882.101} C_VEL
LIN {X 0,Y 383.216,Z 383.372,A -85,B 0,C 180,E1 -11886.317,E2 -11886.317} C_VEL
LIN {X 0,Y 383.13,Z 383.378,A -85,B 0,C 180,E1 -11889.502,E2 -11889.502} C_VEL
LIN {X 0,Y 383.121,Z 383.383,A -85,B 0,C 180,E1 -11893.538,E2 -11893.538} C_VEL
LIN {X 0,Y 383.016,Z 383.402,A -85,B 0,C 180,E1 -11897.42,E2 -11897.42} C_VEL
LIN {X 0,Y 383.005,Z 383.399,A -85,B 0,C 180,E1 -11900.64,E2 -11900.64} C_VEL
LIN {X 0,Y 383,Z 383.401,A -85,B 0,C 180,E1 -11903.809,E2 -11903.809} C_VEL
LIN {X 0,Y 382.962,Z 383.404,A -85,B 0,C 180,E1 -11907.309,E2 -11907.309} C_VEL
LIN {X 0,Y 382.974,Z 383.404,A -85,B 0,C 180,E1 -11910.919,E2 -11910.919} C_VEL
LIN {X 0,Y 383.005,Z 383.396,A -85,B 0,C 180,E1 -11914.669,E2 -11914.669} C_VEL
LIN {X 0,Y 382.985,Z 383.396,A -85,B 0,C 180,E1 -11917.902,E2 -11917.902} C_VEL
LIN {X 0,Y 382.955,Z 383.407,A -85,B 0,C 180,E1 -11921.351,E2 -11921.351} C_VEL
LIN {X 0,Y 382.983,Z 383.404,A -85,B 0,C 180,E1 -11924.302,E2 -11924.302} C_VEL
LIN {X 0,Y 382.977,Z 383.407,A -85,B 0,C 180,E1 -11927.236,E2 -11927.236} C_VEL
LIN {X 0,Y 382.985,Z 383.455,A -85,B 0,C 180,E1 -11930.708,E2 -11930.708} C_VEL
LIN {X 0,Y 387.275,Z 398.765,A -85,B 0,C 180,E1 -11933.418,E2 -11933.418} C_VEL
LIN {X 0,Y 390.92,Z 412.965,A -85,B 0,C 180,E1 -11935.791,E2 -11935.791} C_VEL
LIN {X 0,Y 392.163,Z 418.739,A -85,B 0,C 180,E1 -11936.713,E2 -11936.713} C_VEL
LIN {X 0,Y 389.681,Z 446.662,A -85,B 0,C 180,E1 -11940.576,E2 -11940.576} C_VEL
LIN {X 0,Y 389.409,Z 449.601,A -85,B 0,C 180,E1 -11940.979,E2 -11940.979} C_VEL
LIN {X 0,Y 396.517,Z 502.573,A -85,B 0,C 180,E1 -11942.5,E2 -11942.5} C_VEL
LIN {X 0,Y 394.306,Z 615.666,A -85,B 0,C 180,E1 -11944.568,E2 -11944.568} C_VEL
LIN {X 0,Y 393.571,Z 631.599,A -85,B 0,C 180,E1 -11945.012,E2 -11945.012} C_VEL
LIN {X 0,Y 392.506,Z 646.181,A -85,B 0,C 180,E1 -11945.61,E2 -11945.61} C_VEL
LIN {X 0,Y 391.156,Z 660.51,A -85,B 0,C 180,E1 -11946.395,E2 -11946.395} C_VEL
LIN {X 0,Y 389.785,Z 673.908,A -85,B 0,C 180,E1 -11947.332,E2 -11947.332} C_VEL
LIN {X 0,Y 388.237,Z 687.365,A -85,B 0,C 180,E1 -11948.496,E2 -11948.496} C_VEL
LIN {X 0,Y 386.817,Z 699.804,A -85,B 0,C 180,E1 -11949.806,E2 -11949.806} C_VEL
LIN {X 0,Y 385.518,Z 711.5,A -85,B 0,C 180,E1 -11951.282,E2 -11951.282} C_VEL
LIN {X 0,Y 384.306,Z 722.763,A -85,B 0,C 180,E1 -11952.986,E2 -11952.986} C_VEL
LIN {X 0,Y 383.329,Z 733.034,A -85,B 0,C 180,E1 -11954.855,E2 -11954.855} C_VEL
LIN {X 0,Y 382.664,Z 741.721,A -85,B 0,C 180,E1 -11956.754,E2 -11956.754} C_VEL
LIN {X 0,Y 382.318,Z 749.668,A -85,B 0,C 180,E1 -11958.871,E2 -11958.871} C_VEL
LIN {X 0,Y 382.228,Z 756.084,A -85,B 0,C 180,E1 -11961.008,E2 -11961.008} C_VEL
LIN {X 0,Y 382.319,Z 760.839,A -85,B 0,C 180,E1 -11963.051,E2 -11963.051} C_VEL
LIN {X 0,Y 382.43,Z 763.825,A -85,B 0,C 180,E1 -11964.728,E2 -11964.728} C_VEL
LIN {X 0,Y 382.509,Z 766.447,A -85,B 0,C 180,E1 -11966.84,E2 -11966.84} C_VEL
LIN {X 0,Y 382.77,Z 767.806,A -85,B 0,C 180,E1 -11968.948,E2 -11968.948} C_VEL
LIN {X 0,Y 382.767,Z 767.9,A -85,B 0,C 180,E1 -11971.052,E2 -11971.052} C_VEL
LIN {X 0,Y 382.483,Z 766.759,A -85,B 0,C 180,E1 -11973.159,E2 -11973.159} C_VEL
LIN {X 0,Y 382.511,Z 765.762,A -85,B 0,C 180,E1 -11974.214,E2 -11974.214} C_VEL
LIN {X 0,Y 382.3,Z 762.81,A -85,B 0,C 180,E1 -11976.332,E2 -11976.332} C_VEL
LIN {X 0,Y 382.156,Z 758.571,A -85,B 0,C 180,E1 -11978.46,E2 -11978.46} C_VEL
LIN {X 0,Y 382.184,Z 752.947,A -85,B 0,C 180,E1 -11980.596,E2 -11980.596} C_VEL
LIN {X 0,Y 382.491,Z 745.864,A -85,B 0,C 180,E1 -11982.737,E2 -11982.737} C_VEL
LIN {X 0,Y 383.244,Z 737.162,A -85,B 0,C 180,E1 -11984.876,E2 -11984.876} C_VEL
LIN {X 0,Y 384.25,Z 727.959,A -85,B 0,C 180,E1 -11986.742,E2 -11986.742} C_VEL
LIN {X 0,Y 385.595,Z 716.986,A -85,B 0,C 180,E1 -11988.6,E2 -11988.6} C_VEL
LIN {X 0,Y 387.237,Z 704.809,A -85,B 0,C 180,E1 -11990.309,E2 -11990.309} C_VEL
LIN {X 0,Y 388.879,Z 692.469,A -85,B 0,C 180,E1 -11991.745,E2 -11991.745} C_VEL
LIN {X 0,Y 390.773,Z 679.016,A -85,B 0,C 180,E1 -11993.026,E2 -11993.026} C_VEL
LIN {X 0,Y 392.571,Z 664.598,A -85,B 0,C 180,E1 -11994.138,E2 -11994.138} C_VEL
LIN {X 0,Y 394.214,Z 650.647,A -85,B 0,C 180,E1 -11994.979,E2 -11994.979} C_VEL
LIN {X 0,Y 395.66,Z 635.894,A -85,B 0,C 180,E1 -11995.655,E2 -11995.655} C_VEL
LIN {X 0,Y 396.769,Z 620.826,A -85,B 0,C 180,E1 -11996.142,E2 -11996.142} C_VEL
LIN {X 0,Y 397.414,Z 599.169,A -85,B 0,C 180,E1 -11996.591,E2 -11996.591} C_VEL
LIN {X 0,Y 399.554,Z 503.246,A -85,B 0,C 180,E1 -11998.367,E2 -11998.367} C_VEL
LIN {X 0,Y 396.017,Z 475.787,A -85,B 0,C 180,E1 -11999.235,E2 -11999.235} C_VEL
LIN {X 0,Y 391.32,Z 447.7,A -85,B 0,C 180,E1 -12000.259,E2 -12000.259} C_VEL
LIN {X 0,Y 394.082,Z 422.808,A -85,B 0,C 180,E1 -12003.827,E2 -12003.827} C_VEL
LIN {X 0,Y 392.814,Z 416.419,A -85,B 0,C 180,E1 -12004.925,E2 -12004.925} C_VEL
LIN {X 0,Y 390.076,Z 406.269,A -85,B 0,C 180,E1 -12006.791,E2 -12006.791} C_VEL
LIN {X 0,Y 385.714,Z 391.854,A -85,B 0,C 180,E1 -12009.621,E2 -12009.621} C_VEL
LIN {X 0,Y 382.968,Z 383.404,A -85,B 0,C 180,E1 -12011.435,E2 -12011.435} C_VEL
LIN {X 0,Y 382.984,Z 383.395,A -85,B 0,C 180,E1 -12014.302,E2 -12014.302} C_VEL
LIN {X 0,Y 382.973,Z 383.403,A -85,B 0,C 180,E1 -12017.235,E2 -12017.235} C_VEL
LIN {X 0,Y 382.975,Z 383.403,A -85,B 0,C 180,E1 -12020.418,E2 -12020.418} C_VEL
LIN {X 0,Y 383.002,Z 383.398,A -85,B 0,C 180,E1 -12024.042,E2 -12024.042} C_VEL
LIN {X 0,Y 382.974,Z 383.404,A -85,B 0,C 180,E1 -12027.578,E2 -12027.578} C_VEL
LIN {X 0,Y 382.964,Z 383.407,A -85,B 0,C 180,E1 -12030.298,E2 -12030.298} C_VEL
LIN {X 0,Y 382.991,Z 383.406,A -85,B 0,C 180,E1 -12034.045,E2 -12034.045} C_VEL
LIN {X 0,Y 382.971,Z 383.407,A -85,B 0,C 180,E1 -12037.333,E2 -12037.333} C_VEL
LIN {X 0,Y 382.999,Z 383.405,A -85,B 0,C 180,E1 -12040.713,E2 -12040.713} C_VEL
LIN {X 0,Y 382.995,Z 383.403,A -85,B 0,C 180,E1 -12044.023,E2 -12044.023} C_VEL
LIN {X 0,Y 383.117,Z 383.386,A -85,B 0,C 180,E1 -12047.284,E2 -12047.284} C_VEL
LIN {X 0,Y 383.125,Z 383.383,A -85,B 0,C 180,E1 -12050.497,E2 -12050.497} C_VEL
LIN {X 0,Y 383.215,Z 383.367,A -85,B 0,C 180,E1 -12053.683,E2 -12053.683} C_VEL
LIN {X 0,Y 383.362,Z 383.348,A -85,B 0,C 180,E1 -12057.899,E2 -12057.899} C_VEL
LIN {X 0,Y 383.36,Z 383.351,A -85,B 0,C 180,E1 -12062.102,E2 -12062.102} C_VEL
LIN {X 0,Y 383.219,Z 383.346,A -85,B 0,C 180,E1 -12066.698,E2 -12066.698} C_VEL
LIN {X 0,Y 383.127,Z 383.381,A -85,B 0,C 180,E1 -12069.503,E2 -12069.503} C_VEL
LIN {X 0,Y 383.114,Z 383.368,A -85,B 0,C 180,E1 -12073.537,E2 -12073.537} C_VEL
LIN {X 0,Y 383.083,Z 383.392,A -85,B 0,C 180,E1 -12077.07,E2 -12077.07} C_VEL
LIN {X 0,Y 383.018,Z 383.379,A -85,B 0,C 180,E1 -12080.647,E2 -12080.647} C_VEL
LIN {X 0,Y 382.997,Z 383.401,A -85,B 0,C 180,E1 -12083.81,E2 -12083.81} C_VEL
LIN {X 0,Y 382.96,Z 383.393,A -85,B 0,C 180,E1 -12087.31,E2 -12087.31} C_VEL
LIN {X 0,Y 382.972,Z 383.398,A -85,B 0,C 180,E1 -12090.92,E2 -12090.92} C_VEL
LIN {X 0,Y 383.003,Z 383.407,A -85,B 0,C 180,E1 -12094.67,E2 -12094.67} C_VEL
LIN {X 0,Y 382.987,Z 383.402,A -85,B 0,C 180,E1 -12097.904,E2 -12097.904} C_VEL
LIN {X 0,Y 382.954,Z 383.403,A -85,B 0,C 180,E1 -12101.352,E2 -12101.352} C_VEL
LIN {X 0,Y 382.983,Z 383.394,A -85,B 0,C 180,E1 -12104.303,E2 -12104.303} C_VEL
LIN {X 0,Y 383.006,Z 383.395,A -85,B 0,C 180,E1 -12107.241,E2 -12107.241} C_VEL
LIN {X 0,Y 383.013,Z 383.543,A -85,B 0,C 180,E1 -12110.557,E2 -12110.557} C_VEL
LIN {X 0,Y 384.088,Z 386.415,A -85,B 0,C 180,E1 -12110.731,E2 -12110.731} C_VEL
LIN {X 0,Y 385.634,Z 388.806,A -85,B 0,C 180,E1 -12110.94,E2 -12110.94} C_VEL
LIN {X 0,Y 394.933,Z 405.097,A -85,B 0,C 180,E1 -12112.196,E2 -12112.196} C_VEL
LIN {X 0,Y 401.11,Z 416.963,A -85,B 0,C 180,E1 -12113.009,E2 -12113.009} C_VEL
LIN {X 0,Y 399.161,Z 507.85,A -85,B 0,C 180,E1 -12114.711,E2 -12114.711} C_VEL
LIN {X 0,Y 398.916,Z 523.125,A -85,B 0,C 180,E1 -12115.11,E2 -12115.11} C_VEL
LIN {X 0,Y 398.364,Z 537.051,A -85,B 0,C 180,E1 -12115.656,E2 -12115.656} C_VEL
LIN {X 0,Y 397.405,Z 551.783,A -85,B 0,C 180,E1 -12116.434,E2 -12116.434} C_VEL
LIN {X 0,Y 396.285,Z 565.846,A -85,B 0,C 180,E1 -12117.407,E2 -12117.407} C_VEL
LIN {X 0,Y 395.155,Z 577.044,A -85,B 0,C 180,E1 -12118.356,E2 -12118.356} C_VEL
LIN {X 0,Y 393.52,Z 590.221,A -85,B 0,C 180,E1 -12119.701,E2 -12119.701} C_VEL
LIN {X 0,Y 392.084,Z 601.143,A -85,B 0,C 180,E1 -12121.056,E2 -12121.056} C_VEL
LIN {X 0,Y 390.46,Z 612.091,A -85,B 0,C 180,E1 -12122.68,E2 -12122.68} C_VEL
LIN {X 0,Y 389.016,Z 621.275,A -85,B 0,C 180,E1 -12124.306,E2 -12124.306} C_VEL
LIN {X 0,Y 387.58,Z 630.165,A -85,B 0,C 180,E1 -12126.206,E2 -12126.206} C_VEL
LIN {X 0,Y 386.312,Z 637.464,A -85,B 0,C 180,E1 -12128.098,E2 -12128.098} C_VEL
LIN {X 0,Y 385.236,Z 644.203,A -85,B 0,C 180,E1 -12130.276,E2 -12130.276} C_VEL
LIN {X 0,Y 384.374,Z 649.399,A -85,B 0,C 180,E1 -12132.442,E2 -12132.442} C_VEL
LIN {X 0,Y 383.855,Z 652.366,A -85,B 0,C 180,E1 -12134.061,E2 -12134.061} C_VEL
LIN {X 0,Y 383.344,Z 655.388,A -85,B 0,C 180,E1 -12136.331,E2 -12136.331} C_VEL
LIN {X 0,Y 383.117,Z 656.999,A -85,B 0,C 180,E1 -12138.359,E2 -12138.359} C_VEL
LIN {X 0,Y 383.015,Z 657.559,A -85,B 0,C 180,E1 -12140.495,E2 -12140.495} C_VEL
LIN {X 0,Y 383.03,Z 656.999,A -85,B 0,C 180,E1 -12142.621,E2 -12142.621} C_VEL
LIN {X 0,Y 383.092,Z 655.361,A -85,B 0,C 180,E1 -12144.738,E2 -12144.738} C_VEL
LIN {X 0,Y 383.406,Z 652.582,A -85,B 0,C 180,E1 -12146.848,E2 -12146.848} C_VEL
LIN {X 0,Y 383.746,Z 648.646,A -85,B 0,C 180,E1 -12148.951,E2 -12148.951} C_VEL
LIN {X 0,Y 384.379,Z 643.417,A -85,B 0,C 180,E1 -12151.048,E2 -12151.048} C_VEL
LIN {X 0,Y 385.298,Z 636.753,A -85,B 0,C 180,E1 -12153.137,E2 -12153.137} C_VEL
LIN {X 0,Y 386.311,Z 628.481,A -85,B 0,C 180,E1 -12155.219,E2 -12155.219} C_VEL
LIN {X 0,Y 387.459,Z 619.693,A -85,B 0,C 180,E1 -12157.033,E2 -12157.033} C_VEL
LIN {X 0,Y 388.174,Z 614.217,A -85,B 0,C 180,E1 -12158.005,E2 -12158.005} C_VEL
LIN {X 0,Y 388.011,Z 610.42,A -85,B 0,C 180,E1 -12158.67,E2 -12158.67} C_VEL
LIN {X 0,Y 386.068,Z 604.203,A -85,B 0,C 180,E1 -12159.781,E2 -12159.781} C_VEL
LIN {X 0,Y 384.107,Z 597.639,A -85,B 0,C 180,E1 -12160.848,E2 -12160.848} C_VEL
LIN {X 0,Y 383.907,Z 593.241,A -85,B 0,C 180,E1 -12161.436,E2 -12161.436} C_VEL
LIN {X 0,Y 385.202,Z 580.912,A -85,B 0,C 180,E1 -12162.781,E2 -12162.781} C_VEL
LIN {X 0,Y 386.487,Z 567.839,A -85,B 0,C 180,E1 -12163.942,E2 -12163.942} C_VEL
LIN {X 0,Y 387.624,Z 553.364,A -85,B 0,C 180,E1 -12164.973,E2 -12164.973} C_VEL
LIN {X 0,Y 388.442,Z 539.356,A -85,B 0,C 180,E1 -12165.747,E2 -12165.747} C_VEL
LIN {X 0,Y 388.983,Z 524.013,A -85,B 0,C 180,E1 -12166.377,E2 -12166.377} C_VEL
LIN {X 0,Y 389.201,Z 508.528,A -85,B 0,C 180,E1 -12166.793,E2 -12166.793} C_VEL
LIN {X 0,Y 390.882,Z 416.166,A -85,B 0,C 180,E1 -12168.523,E2 -12168.523} C_VEL
LIN {X 0,Y 380.008,Z 393.091,A -85,B 0,C 180,E1 -12169.79,E2 -12169.79} C_VEL
LIN {X 0,Y 376.191,Z 385.26,A -85,B 0,C 180,E1 -12170.249,E2 -12170.249} C_VEL
LIN {X 0,Y 375.996,Z 384.274,A -85,B 0,C 180,E1 -12170.311,E2 -12170.311} C_VEL
LIN {X 0,Y 375.968,Z 384.279,A -85,B 0,C 180,E1 -12173.657,E2 -12173.657} C_VEL
LIN {X 0,Y 375.91,Z 384.286,A -85,B 0,C 180,E1 -12176.66,E2 -12176.66} C_VEL
LIN {X 0,Y 375.912,Z 384.275,A -85,B 0,C 180,E1 -12179.084,E2 -12179.084} C_VEL
LIN {X 0,Y 375.953,Z 384.28,A -85,B 0,C 180,E1 -12181.562,E2 -12181.562} C_VEL
LIN {X 0,Y 375.947,Z 384.281,A -85,B 0,C 180,E1 -12185.416,E2 -12185.416} C_VEL
LIN {X 0,Y 375.932,Z 384.281,A -85,B 0,C 180,E1 -12188.262,E2 -12188.262} C_VEL
LIN {X 0,Y 375.907,Z 384.286,A -85,B 0,C 180,E1 -12191.595,E2 -12191.595} C_VEL
LIN {X 0,Y 375.907,Z 384.288,A -85,B 0,C 180,E1 -12195.271,E2 -12195.271} C_VEL
LIN {X 0,Y 375.91,Z 384.28,A -85,B 0,C 180,E1 -12198.402,E2 -12198.402} C_VEL
LIN {X 0,Y 375.948,Z 384.275,A -85,B 0,C 180,E1 -12201.909,E2 -12201.909} C_VEL
LIN {X 0,Y 375.97,Z 384.274,A -85,B 0,C 180,E1 -12205.333,E2 -12205.333} C_VEL
LIN {X 0,Y 375.93,Z 384.282,A -85,B 0,C 180,E1 -12208.435,E2 -12208.435} C_VEL
LIN {X 0,Y 375.941,Z 384.277,A -85,B 0,C 180,E1 -12211.476,E2 -12211.476} C_VEL
LIN {X 0,Y 375.942,Z 384.279,A -85,B 0,C 180,E1 -12214.534,E2 -12214.534} C_VEL
LIN {X 0,Y 375.948,Z 384.279,A -85,B 0,C 180,E1 -12218.044,E2 -12218.044} C_VEL
LIN {X 0,Y 375.996,Z 384.268,A -85,B 0,C 180,E1 -12221.472,E2 -12221.472} C_VEL
LIN {X 0,Y 376.047,Z 384.266,A -85,B 0,C 180,E1 -12224.832,E2 -12224.832} C_VEL
LIN {X 0,Y 376.037,Z 384.238,A -85,B 0,C 180,E1 -12228.136,E2 -12228.136} C_VEL
LIN {X 0,Y 376.179,Z 384.24,A -85,B 0,C 180,E1 -12231.955,E2 -12231.955} C_VEL
LIN {X 0,Y 376.131,Z 384.255,A -85,B 0,C 180,E1 -12234.639,E2 -12234.639} C_VEL
LIN {X 0,Y 376.32,Z 384.223,A -85,B 0,C 180,E1 -12237.859,E2 -12237.859} C_VEL
LIN {X 0,Y 376.331,Z 384.226,A -85,B 0,C 180,E1 -12242.14,E2 -12242.14} C_VEL
LIN {X 0,Y 376.175,Z 384.249,A -85,B 0,C 180,E1 -12246.436,E2 -12246.436} C_VEL
LIN {X 0,Y 376.101,Z 384.254,A -85,B 0,C 180,E1 -12249.682,E2 -12249.682} C_VEL
LIN {X 0,Y 376.084,Z 384.258,A -85,B 0,C 180,E1 -12253.658,E2 -12253.658} C_VEL
LIN {X 0,Y 375.974,Z 384.277,A -85,B 0,C 180,E1 -12257.577,E2 -12257.577} C_VEL
LIN {X 0,Y 375.972,Z 384.276,A -85,B 0,C 180,E1 -12260.832,E2 -12260.832} C_VEL
LIN {X 0,Y 375.927,Z 384.282,A -85,B 0,C 180,E1 -12264.286,E2 -12264.286} C_VEL
LIN {X 0,Y 375.904,Z 384.28,A -85,B 0,C 180,E1 -12266.661,E2 -12266.661} C_VEL
LIN {X 0,Y 375.906,Z 384.284,A -85,B 0,C 180,E1 -12269.084,E2 -12269.084} C_VEL
LIN {X 0,Y 375.949,Z 384.284,A -85,B 0,C 180,E1 -12271.563,E2 -12271.563} C_VEL
LIN {X 0,Y 375.942,Z 384.279,A -85,B 0,C 180,E1 -12275.417,E2 -12275.417} C_VEL
LIN {X 0,Y 375.927,Z 384.272,A -85,B 0,C 180,E1 -12278.263,E2 -12278.263} C_VEL
LIN {X 0,Y 375.908,Z 384.281,A -85,B 0,C 180,E1 -12281.597,E2 -12281.597} C_VEL
LIN {X 0,Y 375.915,Z 384.282,A -85,B 0,C 180,E1 -12284.73,E2 -12284.73} C_VEL
LIN {X 0,Y 375.903,Z 384.282,A -85,B 0,C 180,E1 -12287.697,E2 -12287.697} C_VEL
LIN {X 0,Y 375.941,Z 384.36,A -85,B 0,C 180,E1 -12290.241,E2 -12290.241} C_VEL
LIN {X 0,Y 380.124,Z 399.165,A -85,B 0,C 180,E1 -12292.932,E2 -12292.932} C_VEL
LIN {X 0,Y 383.932,Z 413.926,A -85,B 0,C 180,E1 -12295.461,E2 -12295.461} C_VEL
LIN {X 0,Y 385.36,Z 420.384,A -85,B 0,C 180,E1 -12296.518,E2 -12296.518} C_VEL
LIN {X 0,Y 382.735,Z 448.432,A -85,B 0,C 180,E1 -12300.468,E2 -12300.468} C_VEL
LIN {X 0,Y 390.019,Z 503.397,A -85,B 0,C 180,E1 -12302.097,E2 -12302.097} C_VEL
LIN {X 0,Y 387.688,Z 616.89,A -85,B 0,C 180,E1 -12304.21,E2 -12304.21} C_VEL
LIN {X 0,Y 386.918,Z 631.955,A -85,B 0,C 180,E1 -12304.66,E2 -12304.66} C_VEL
LIN {X 0,Y 385.757,Z 646.806,A -85,B 0,C 180,E1 -12305.299,E2 -12305.299} C_VEL
LIN {X 0,Y 384.371,Z 660.743,A -85,B 0,C 180,E1 -12306.095,E2 -12306.095} C_VEL
LIN {X 0,Y 382.945,Z 673.89,A -85,B 0,C 180,E1 -12307.046,E2 -12307.046} C_VEL
LIN {X 0,Y 381.375,Z 687.174,A -85,B 0,C 180,E1 -12308.231,E2 -12308.231} C_VEL
LIN {X 0,Y 379.747,Z 700.572,A -85,B 0,C 180,E1 -12309.696,E2 -12309.696} C_VEL
LIN {X 0,Y 378.467,Z 711.717,A -85,B 0,C 180,E1 -12311.161,E2 -12311.161} C_VEL
LIN {X 0,Y 377.373,Z 721.444,A -85,B 0,C 180,E1 -12312.664,E2 -12312.664} C_VEL
LIN {X 0,Y 376.329,Z 731.768,A -85,B 0,C 180,E1 -12314.566,E2 -12314.566} C_VEL
LIN {X 0,Y 375.61,Z 741.08,A -85,B 0,C 180,E1 -12316.646,E2 -12316.646} C_VEL
LIN {X 0,Y 375.267,Z 748.486,A -85,B 0,C 180,E1 -12318.659,E2 -12318.659} C_VEL
LIN {X 0,Y 375.155,Z 754.934,A -85,B 0,C 180,E1 -12320.837,E2 -12320.837} C_VEL
LIN {X 0,Y 375.266,Z 759.928,A -85,B 0,C 180,E1 -12323.017,E2 -12323.017} C_VEL
LIN {X 0,Y 375.387,Z 762.745,A -85,B 0,C 180,E1 -12324.628,E2 -12324.628} C_VEL
LIN {X 0,Y 375.472,Z 765.394,A -85,B 0,C 180,E1 -12326.781,E2 -12326.781} C_VEL
LIN {X 0,Y 375.743,Z 766.771,A -85,B 0,C 180,E1 -12328.928,E2 -12328.928} C_VEL
LIN {X 0,Y 375.739,Z 766.89,A -85,B 0,C 180,E1 -12331.071,E2 -12331.071} C_VEL
LIN {X 0,Y 375.441,Z 765.77,A -85,B 0,C 180,E1 -12333.219,E2 -12333.219} C_VEL
LIN {X 0,Y 375.471,Z 764.785,A -85,B 0,C 180,E1 -12334.293,E2 -12334.293} C_VEL
LIN {X 0,Y 375.249,Z 761.855,A -85,B 0,C 180,E1 -12336.452,E2 -12336.452} C_VEL
LIN {X 0,Y 375.083,Z 757.623,A -85,B 0,C 180,E1 -12338.62,E2 -12338.62} C_VEL
LIN {X 0,Y 375.121,Z 752.025,A -85,B 0,C 180,E1 -12340.798,E2 -12340.798} C_VEL
LIN {X 0,Y 375.457,Z 744.974,A -85,B 0,C 180,E1 -12342.98,E2 -12342.98} C_VEL
LIN {X 0,Y 376.145,Z 737.472,A -85,B 0,C 180,E1 -12344.886,E2 -12344.886} C_VEL
LIN {X 0,Y 377.167,Z 728.552,A -85,B 0,C 180,E1 -12346.787,E2 -12346.787} C_VEL
LIN {X 0,Y 378.502,Z 718.267,A -85,B 0,C 180,E1 -12348.62,E2 -12348.62} C_VEL
LIN {X 0,Y 380.055,Z 707.106,A -85,B 0,C 180,E1 -12350.286,E2 -12350.286} C_VEL
LIN {X 0,Y 381.693,Z 695.434,A -85,B 0,C 180,E1 -12351.749,E2 -12351.749} C_VEL
LIN {X 0,Y 383.62,Z 682.839,A -85,B 0,C 180,E1 -12353.053,E2 -12353.053} C_VEL
LIN {X 0,Y 385.514,Z 668.679,A -85,B 0,C 180,E1 -12354.25,E2 -12354.25} C_VEL
LIN {X 0,Y 387.232,Z 654.981,A -85,B 0,C 180,E1 -12355.173,E2 -12355.173} C_VEL
LIN {X 0,Y 388.92,Z 640.52,A -85,B 0,C 180,E1 -12355.917,E2 -12355.917} C_VEL
LIN {X 0,Y 390.213,Z 624.9,A -85,B 0,C 180,E1 -12356.507,E2 -12356.507} C_VEL
LIN {X 0,Y 390.923,Z 609.663,A -85,B 0,C 180,E1 -12356.887,E2 -12356.887} C_VEL
LIN {X 0,Y 393.412,Z 504.083,A -85,B 0,C 180,E1 -12358.871,E2 -12358.871} C_VEL
LIN {X 0,Y 389.96,Z 477.131,A -85,B 0,C 180,E1 -12359.745,E2 -12359.745} C_VEL
LIN {X 0,Y 384.902,Z 446.555,A -85,B 0,C 180,E1 -12360.887,E2 -12360.887} C_VEL
LIN {X 0,Y 387.326,Z 425.754,A -85,B 0,C 180,E1 -12363.928,E2 -12363.928} C_VEL
LIN {X 0,Y 387.401,Z 423.858,A -85,B 0,C 180,E1 -12364.219,E2 -12364.219} C_VEL
LIN {X 0,Y 384.396,Z 411.681,A -85,B 0,C 180,E1 -12366.442,E2 -12366.442} C_VEL
LIN {X 0,Y 380.13,Z 397.3,A -85,B 0,C 180,E1 -12369.286,E2 -12369.286} C_VEL
LIN {X 0,Y 375.92,Z 384.283,A -85,B 0,C 180,E1 -12372.103,E2 -12372.103} C_VEL
LIN {X 0,Y 375.911,Z 384.264,A -85,B 0,C 180,E1 -12375.269,E2 -12375.269} C_VEL
LIN {X 0,Y 375.903,Z 384.282,A -85,B 0,C 180,E1 -12378.402,E2 -12378.402} C_VEL
LIN {X 0,Y 375.941,Z 384.278,A -85,B 0,C 180,E1 -12381.909,E2 -12381.909} C_VEL
LIN {X 0,Y 375.964,Z 384.278,A -85,B 0,C 180,E1 -12385.333,E2 -12385.333} C_VEL
LIN {X 0,Y 375.945,Z 384.282,A -85,B 0,C 180,E1 -12388.437,E2 -12388.437} C_VEL
LIN {X 0,Y 375.905,Z 384.285,A -85,B 0,C 180,E1 -12392.134,E2 -12392.134} C_VEL
LIN {X 0,Y 375.924,Z 384.286,A -85,B 0,C 180,E1 -12394.533,E2 -12394.533} C_VEL
LIN {X 0,Y 375.957,Z 384.282,A -85,B 0,C 180,E1 -12396.886,E2 -12396.886} C_VEL
LIN {X 0,Y 375.947,Z 384.282,A -85,B 0,C 180,E1 -12400.337,E2 -12400.337} C_VEL
LIN {X 0,Y 375.945,Z 384.279,A -85,B 0,C 180,E1 -12403.715,E2 -12403.715} C_VEL
LIN {X 0,Y 376.088,Z 384.263,A -85,B 0,C 180,E1 -12407.042,E2 -12407.042} C_VEL
LIN {X 0,Y 376.096,Z 384.257,A -85,B 0,C 180,E1 -12410.318,E2 -12410.318} C_VEL
LIN {X 0,Y 376.175,Z 384.243,A -85,B 0,C 180,E1 -12413.564,E2 -12413.564} C_VEL
LIN {X 0,Y 376.327,Z 384.224,A -85,B 0,C 180,E1 -12417.86,E2 -12417.86} C_VEL
LIN {X 0,Y 376.325,Z 384.228,A -85,B 0,C 180,E1 -12422.141,E2 -12422.141} C_VEL
LIN {X 0,Y 376.183,Z 384.222,A -85,B 0,C 180,E1 -12426.687,E2 -12426.687} C_VEL
LIN {X 0,Y 376.098,Z 384.257,A -85,B 0,C 180,E1 -12429.682,E2 -12429.682} C_VEL
LIN {X 0,Y 376.078,Z 384.242,A -85,B 0,C 180,E1 -12433.658,E2 -12433.658} C_VEL
LIN {X 0,Y 376.021,Z 384.27,A -85,B 0,C 180,E1 -12437.401,E2 -12437.401} C_VEL
LIN {X 0,Y 375.968,Z 384.256,A -85,B 0,C 180,E1 -12440.833,E2 -12440.833} C_VEL
LIN {X 0,Y 375.948,Z 384.281,A -85,B 0,C 180,E1 -12444.285,E2 -12444.285} C_VEL
LIN {X 0,Y 375.908,Z 384.277,A -85,B 0,C 180,E1 -12447.866,E2 -12447.866} C_VEL
LIN {X 0,Y 375.945,Z 384.277,A -85,B 0,C 180,E1 -12450.694,E2 -12450.694} C_VEL
LIN {X 0,Y 375.949,Z 384.282,A -85,B 0,C 180,E1 -12454.113,E2 -12454.113} C_VEL
LIN {X 0,Y 375.941,Z 384.272,A -85,B 0,C 180,E1 -12456.743,E2 -12456.743} C_VEL
LIN {X 0,Y 375.932,Z 384.277,A -85,B 0,C 180,E1 -12459.963,E2 -12459.963} C_VEL
LIN {X 0,Y 375.918,Z 384.274,A -85,B 0,C 180,E1 -12463.768,E2 -12463.768} C_VEL
LIN {X 0,Y 375.928,Z 384.276,A -85,B 0,C 180,E1 -12466.812,E2 -12466.812} C_VEL
LIN {X 0,Y 375.911,Z 384.279,A -85,B 0,C 180,E1 -12469.823,E2 -12469.823} C_VEL
LIN {X 0,Y 376.97,Z 387.198,A -85,B 0,C 180,E1 -12470.005,E2 -12470.005} C_VEL
LIN {X 0,Y 378.42,Z 389.324,A -85,B 0,C 180,E1 -12470.208,E2 -12470.208} C_VEL
LIN {X 0,Y 388.653,Z 407.072,A -85,B 0,C 180,E1 -12471.639,E2 -12471.639} C_VEL
LIN {X 0,Y 395.129,Z 419.47,A -85,B 0,C 180,E1 -12472.519,E2 -12472.519} C_VEL
LIN {X 0,Y 393.07,Z 505.277,A -85,B 0,C 180,E1 -12474.139,E2 -12474.139} C_VEL
LIN {X 0,Y 392.785,Z 522.461,A -85,B 0,C 180,E1 -12474.562,E2 -12474.562} C_VEL
LIN {X 0,Y 392.198,Z 537.281,A -85,B 0,C 180,E1 -12475.133,E2 -12475.133} C_VEL
LIN {X 0,Y 391.293,Z 551.509,A -85,B 0,C 180,E1 -12475.883,E2 -12475.883} C_VEL
LIN {X 0,Y 390.13,Z 565.331,A -85,B 0,C 180,E1 -12476.827,E2 -12476.827} C_VEL
LIN {X 0,Y 388.799,Z 578.42,A -85,B 0,C 180,E1 -12477.945,E2 -12477.945} C_VEL
LIN {X 0,Y 387.104,Z 591.485,A -85,B 0,C 180,E1 -12479.306,E2 -12479.306} C_VEL
LIN {X 0,Y 385.51,Z 602.875,A -85,B 0,C 180,E1 -12480.752,E2 -12480.752} C_VEL
LIN {X 0,Y 383.755,Z 614.041,A -85,B 0,C 180,E1 -12482.458,E2 -12482.458} C_VEL
LIN {X 0,Y 382.036,Z 624.215,A -85,B 0,C 180,E1 -12484.345,E2 -12484.345} C_VEL
LIN {X 0,Y 380.55,Z 632.914,A -85,B 0,C 180,E1 -12486.318,E2 -12486.318} C_VEL
LIN {X 0,Y 379.262,Z 639.917,A -85,B 0,C 180,E1 -12488.248,E2 -12488.248} C_VEL
LIN {X 0,Y 378.159,Z 646.322,A -85,B 0,C 180,E1 -12490.457,E2 -12490.457} C_VEL
LIN {X 0,Y 377.287,Z 651.246,A -85,B 0,C 180,E1 -12492.661,E2 -12492.661} C_VEL
LIN {X 0,Y 376.641,Z 654.842,A -85,B 0,C 180,E1 -12494.857,E2 -12494.857} C_VEL
LIN {X 0,Y 376.242,Z 657.217,A -85,B 0,C 180,E1 -12497.048,E2 -12497.048} C_VEL
LIN {X 0,Y 376.037,Z 658.399,A -85,B 0,C 180,E1 -12499.229,E2 -12499.229} C_VEL
LIN {X 0,Y 375.982,Z 658.452,A -85,B 0,C 180,E1 -12501.4,E2 -12501.4} C_VEL
LIN {X 0,Y 376.068,Z 657.411,A -85,B 0,C 180,E1 -12503.563,E2 -12503.563} C_VEL
LIN {X 0,Y 376.099,Z 655.302,A -85,B 0,C 180,E1 -12505.714,E2 -12505.714} C_VEL
LIN {X 0,Y 376.56,Z 652.001,A -85,B 0,C 180,E1 -12507.861,E2 -12507.861} C_VEL
LIN {X 0,Y 376.999,Z 647.512,A -85,B 0,C 180,E1 -12510,E2 -12510} C_VEL
LIN {X 0,Y 377.855,Z 641.64,A -85,B 0,C 180,E1 -12512.132,E2 -12512.132} C_VEL
LIN {X 0,Y 378.813,Z 634.301,A -85,B 0,C 180,E1 -12514.256,E2 -12514.256} C_VEL
LIN {X 0,Y 379.803,Z 626.452,A -85,B 0,C 180,E1 -12516.108,E2 -12516.108} C_VEL
LIN {X 0,Y 381.141,Z 617.017,A -85,B 0,C 180,E1 -12517.949,E2 -12517.949} C_VEL
LIN {X 0,Y 382.331,Z 607.405,A -85,B 0,C 180,E1 -12519.523,E2 -12519.523} C_VEL
LIN {X 0,Y 383.641,Z 596.002,A -85,B 0,C 180,E1 -12521.09,E2 -12521.09} C_VEL
LIN {X 0,Y 383.907,Z 593.241,A -85,B 0,C 180,E1 -12521.436,E2 -12521.436} C_VEL
LIN {X 0,Y 383.558,Z 590.247,A -85,B 0,C 180,E1 -12521.829,E2 -12521.829} C_VEL
LIN {X 0,Y 379.324,Z 581.023,A -85,B 0,C 180,E1 -12523.167,E2 -12523.167} C_VEL
LIN {X 0,Y 379.011,Z 577.813,A -85,B 0,C 180,E1 -12523.516,E2 -12523.516} C_VEL
LIN {X 0,Y 380.166,Z 565.23,A -85,B 0,C 180,E1 -12524.589,E2 -12524.589} C_VEL
LIN {X 0,Y 381.297,Z 550.791,A -85,B 0,C 180,E1 -12525.57,E2 -12525.57} C_VEL
LIN {X 0,Y 382.138,Z 535.796,A -85,B 0,C 180,E1 -12526.349,E2 -12526.349} C_VEL
LIN {X 0,Y 382.544,Z 520.155,A -85,B 0,C 180,E1 -12526.935,E2 -12526.935} C_VEL
LIN {X 0,Y 382.856,Z 499.203,A -85,B 0,C 180,E1 -12527.405,E2 -12527.405} C_VEL
LIN {X 0,Y 384.457,Z 418.07,A -85,B 0,C 180,E1 -12528.944,E2 -12528.944} C_VEL
LIN {X 0,Y 373.053,Z 394.023,A -85,B 0,C 180,E1 -12530.31,E2 -12530.31} C_VEL
LIN {X 0,Y 369.086,Z 386.013,A -85,B 0,C 180,E1 -12530.802,E2 -12530.802} C_VEL
LIN {X 0,Y 368.954,Z 385.153,A -85,B 0,C 180,E1 -12530.89,E2 -12530.89} C_VEL
LIN {X 0,Y 368.906,Z 385.158,A -85,B 0,C 180,E1 -12533.872,E2 -12533.872} C_VEL
LIN {X 0,Y 368.856,Z 385.167,A -85,B 0,C 180,E1 -12537.212,E2 -12537.212} C_VEL
LIN {X 0,Y 368.891,Z 385.143,A -85,B 0,C 180,E1 -12539.692,E2 -12539.692} C_VEL
LIN {X 0,Y 368.895,Z 385.16,A -85,B 0,C 180,E1 -12543.042,E2 -12543.042} C_VEL
LIN {X 0,Y 368.909,Z 385.154,A -85,B 0,C 180,E1 -12546.197,E2 -12546.197} C_VEL
LIN {X 0,Y 368.871,Z 385.163,A -85,B 0,C 180,E1 -12548.956,E2 -12548.956} C_VEL
LIN {X 0,Y 368.851,Z 385.162,A -85,B 0,C 180,E1 -12552.004,E2 -12552.004} C_VEL
LIN {X 0,Y 368.858,Z 385.165,A -85,B 0,C 180,E1 -12555.172,E2 -12555.172} C_VEL
LIN {X 0,Y 368.857,Z 385.159,A -85,B 0,C 180,E1 -12558.174,E2 -12558.174} C_VEL
LIN {X 0,Y 368.872,Z 385.158,A -85,B 0,C 180,E1 -12561.366,E2 -12561.366} C_VEL
LIN {X 0,Y 368.926,Z 385.154,A -85,B 0,C 180,E1 -12565.145,E2 -12565.145} C_VEL
LIN {X 0,Y 368.892,Z 385.162,A -85,B 0,C 180,E1 -12569.043,E2 -12569.043} C_VEL
LIN {X 0,Y 368.901,Z 385.155,A -85,B 0,C 180,E1 -12571.557,E2 -12571.557} C_VEL
LIN {X 0,Y 368.916,Z 385.152,A -85,B 0,C 180,E1 -12575.221,E2 -12575.221} C_VEL
LIN {X 0,Y 368.914,Z 385.157,A -85,B 0,C 180,E1 -12578.98,E2 -12578.98} C_VEL
LIN {X 0,Y 368.985,Z 385.142,A -85,B 0,C 180,E1 -12582.257,E2 -12582.257} C_VEL
LIN {X 0,Y 369.031,Z 385.13,A -85,B 0,C 180,E1 -12586.228,E2 -12586.228} C_VEL
LIN {X 0,Y 369.051,Z 385.106,A -85,B 0,C 180,E1 -12590.131,E2 -12590.131} C_VEL
LIN {X 0,Y 369.146,Z 385.124,A -85,B 0,C 180,E1 -12593.44,E2 -12593.44} C_VEL
LIN {X 0,Y 369.283,Z 385.099,A -85,B 0,C 180,E1 -12597.818,E2 -12597.818} C_VEL
LIN {X 0,Y 369.295,Z 385.103,A -85,B 0,C 180,E1 -12602.181,E2 -12602.181} C_VEL
LIN {X 0,Y 369.136,Z 385.125,A -85,B 0,C 180,E1 -12606.559,E2 -12606.559} C_VEL
LIN {X 0,Y 369.051,Z 385.133,A -85,B 0,C 180,E1 -12609.868,E2 -12609.868} C_VEL
LIN {X 0,Y 369.031,Z 385.135,A -85,B 0,C 180,E1 -12613.772,E2 -12613.772} C_VEL
LIN {X 0,Y 368.929,Z 385.152,A -85,B 0,C 180,E1 -12617.746,E2 -12617.746} C_VEL
LIN {X 0,Y 368.902,Z 385.159,A -85,B 0,C 180,E1 -12621.221,E2 -12621.221} C_VEL
LIN {X 0,Y 368.901,Z 385.158,A -85,B 0,C 180,E1 -12623.874,E2 -12623.874} C_VEL
LIN {X 0,Y 368.851,Z 385.161,A -85,B 0,C 180,E1 -12627.212,E2 -12627.212} C_VEL
LIN {X 0,Y 368.886,Z 385.159,A -85,B 0,C 180,E1 -12629.693,E2 -12629.693} C_VEL
LIN {X 0,Y 368.89,Z 385.151,A -85,B 0,C 180,E1 -12633.043,E2 -12633.043} C_VEL
LIN {X 0,Y 368.904,Z 385.161,A -85,B 0,C 180,E1 -12636.198,E2 -12636.198} C_VEL
LIN {X 0,Y 368.867,Z 385.152,A -85,B 0,C 180,E1 -12638.957,E2 -12638.957} C_VEL
LIN {X 0,Y 368.853,Z 385.157,A -85,B 0,C 180,E1 -12642.005,E2 -12642.005} C_VEL
LIN {X 0,Y 368.867,Z 385.158,A -85,B 0,C 180,E1 -12645.175,E2 -12645.175} C_VEL
LIN {X 0,Y 368.855,Z 385.151,A -85,B 0,C 180,E1 -12648.175,E2 -12648.175} C_VEL
LIN {X 0,Y 368.881,Z 385.15,A -85,B 0,C 180,E1 -12649.741,E2 -12649.741} C_VEL
LIN {X 0,Y 373.342,Z 400.996,A -85,B 0,C 180,E1 -12652.687,E2 -12652.687} C_VEL
LIN {X 0,Y 377.201,Z 415.962,A -85,B 0,C 180,E1 -12655.304,E2 -12655.304} C_VEL
LIN {X 0,Y 378.537,Z 422.201,A -85,B 0,C 180,E1 -12656.342,E2 -12656.342} C_VEL
LIN {X 0,Y 376.047,Z 447.545,A -85,B 0,C 180,E1 -12659.981,E2 -12659.981} C_VEL
LIN {X 0,Y 383.515,Z 503.857,A -85,B 0,C 180,E1 -12661.671,E2 -12661.671} C_VEL
LIN {X 0,Y 381.138,Z 616.533,A -85,B 0,C 180,E1 -12663.807,E2 -12663.807} C_VEL
LIN {X 0,Y 380.276,Z 632.266,A -85,B 0,C 180,E1 -12664.296,E2 -12664.296} C_VEL
LIN {X 0,Y 379.007,Z 647.393,A -85,B 0,C 180,E1 -12664.975,E2 -12664.975} C_VEL
LIN {X 0,Y 377.425,Z 662.417,A -85,B 0,C 180,E1 -12665.879,E2 -12665.879} C_VEL
LIN {X 0,Y 375.746,Z 677.069,A -85,B 0,C 180,E1 -12667.018,E2 -12667.018} C_VEL
LIN {X 0,Y 374.011,Z 690.891,A -85,B 0,C 180,E1 -12668.36,E2 -12668.36} C_VEL
LIN {X 0,Y 372.515,Z 703.517,A -85,B 0,C 180,E1 -12669.86,E2 -12669.86} C_VEL
LIN {X 0,Y 371.056,Z 715.039,A -85,B 0,C 180,E1 -12671.503,E2 -12671.503} C_VEL
LIN {X 0,Y 369.815,Z 726.262,A -85,B 0,C 180,E1 -12673.437,E2 -12673.437} C_VEL
LIN {X 0,Y 368.957,Z 735.637,A -85,B 0,C 180,E1 -12675.381,E2 -12675.381} C_VEL
LIN {X 0,Y 368.375,Z 743.437,A -85,B 0,C 180,E1 -12677.326,E2 -12677.326} C_VEL
LIN {X 0,Y 368.107,Z 750.725,A -85,B 0,C 180,E1 -12679.55,E2 -12679.55} C_VEL
LIN {X 0,Y 368.137,Z 756.462,A -85,B 0,C 180,E1 -12681.768,E2 -12681.768} C_VEL
LIN {X 0,Y 368.218,Z 759.824,A -85,B 0,C 180,E1 -12683.424,E2 -12683.424} C_VEL
LIN {X 0,Y 368.436,Z 763.171,A -85,B 0,C 180,E1 -12685.624,E2 -12685.624} C_VEL
LIN {X 0,Y 368.477,Z 765.175,A -85,B 0,C 180,E1 -12687.813,E2 -12687.813} C_VEL
LIN {X 0,Y 368.715,Z 765.735,A -85,B 0,C 180,E1 -12688.907,E2 -12688.907} C_VEL
LIN {X 0,Y 368.71,Z 765.879,A -85,B 0,C 180,E1 -12691.092,E2 -12691.092} C_VEL
LIN {X 0,Y 368.4,Z 764.782,A -85,B 0,C 180,E1 -12693.28,E2 -12693.28} C_VEL
LIN {X 0,Y 368.412,Z 763.807,A -85,B 0,C 180,E1 -12694.376,E2 -12694.376} C_VEL
LIN {X 0,Y 368.199,Z 760.902,A -85,B 0,C 180,E1 -12696.576,E2 -12696.576} C_VEL
LIN {X 0,Y 368.002,Z 756.676,A -85,B 0,C 180,E1 -12698.788,E2 -12698.788} C_VEL
LIN {X 0,Y 368.06,Z 751.108,A -85,B 0,C 180,E1 -12701.007,E2 -12701.007} C_VEL
LIN {X 0,Y 368.533,Z 743.345,A -85,B 0,C 180,E1 -12703.449,E2 -12703.449} C_VEL
LIN {X 0,Y 369.304,Z 735.466,A -85,B 0,C 180,E1 -12705.451,E2 -12705.451} C_VEL
LIN {X 0,Y 370.438,Z 726.357,A -85,B 0,C 180,E1 -12707.385,E2 -12707.385} C_VEL
LIN {X 0,Y 371.728,Z 717.154,A -85,B 0,C 180,E1 -12709.036,E2 -12709.036} C_VEL
LIN {X 0,Y 373.311,Z 706.432,A -85,B 0,C 180,E1 -12710.669,E2 -12710.669} C_VEL
LIN {X 0,Y 375.028,Z 694.842,A -85,B 0,C 180,E1 -12712.156,E2 -12712.156} C_VEL
LIN {X 0,Y 377.016,Z 682.342,A -85,B 0,C 180,E1 -12713.48,E2 -12713.48} C_VEL
LIN {X 0,Y 379.031,Z 668.318,A -85,B 0,C 180,E1 -12714.693,E2 -12714.693} C_VEL
LIN {X 0,Y 380.98,Z 653.72,A -85,B 0,C 180,E1 -12715.689,E2 -12715.689} C_VEL
LIN {X 0,Y 382.683,Z 639.21,A -85,B 0,C 180,E1 -12716.445,E2 -12716.445} C_VEL
LIN {X 0,Y 384.045,Z 623.471,A -85,B 0,C 180,E1 -12717.04,E2 -12717.04} C_VEL
LIN {X 0,Y 384.784,Z 608.032,A -85,B 0,C 180,E1 -12717.426,E2 -12717.426} C_VEL
LIN {X 0,Y 387.307,Z 504.744,A -85,B 0,C 180,E1 -12719.396,E2 -12719.396} C_VEL
LIN {X 0,Y 383.897,Z 478.158,A -85,B 0,C 180,E1 -12720.283,E2 -12720.283} C_VEL
LIN {X 0,Y 379.043,Z 448.573,A -85,B 0,C 180,E1 -12721.406,E2 -12721.406} C_VEL
LIN {X 0,Y 378.479,Z 445.447,A -85,B 0,C 180,E1 -12721.537,E2 -12721.537} C_VEL
LIN {X 0,Y 380.778,Z 426.199,A -85,B 0,C 180,E1 -12724.417,E2 -12724.417} C_VEL
LIN {X 0,Y 378.105,Z 414.972,A -85,B 0,C 180,E1 -12726.497,E2 -12726.497} C_VEL
LIN {X 0,Y 373.659,Z 399.862,A -85,B 0,C 180,E1 -12729.543,E2 -12729.543} C_VEL
LIN {X 0,Y 368.89,Z 385.156,A -85,B 0,C 180,E1 -12732.789,E2 -12732.789} C_VEL
LIN {X 0,Y 368.873,Z 385.149,A -85,B 0,C 180,E1 -12736.694,E2 -12736.694} C_VEL
LIN {X 0,Y 368.875,Z 385.16,A -85,B 0,C 180,E1 -12739.647,E2 -12739.647} C_VEL
LIN {X 0,Y 368.885,Z 385.158,A -85,B 0,C 180,E1 -12743.145,E2 -12743.145} C_VEL
LIN {X 0,Y 368.884,Z 385.157,A -85,B 0,C 180,E1 -12746.461,E2 -12746.461} C_VEL
LIN {X 0,Y 368.902,Z 385.154,A -85,B 0,C 180,E1 -12749.044,E2 -12749.044} C_VEL
LIN {X 0,Y 368.895,Z 385.161,A -85,B 0,C 180,E1 -12751.557,E2 -12751.557} C_VEL
LIN {X 0,Y 368.907,Z 385.16,A -85,B 0,C 180,E1 -12754.013,E2 -12754.013} C_VEL
LIN {X 0,Y 368.883,Z 385.162,A -85,B 0,C 180,E1 -12757.602,E2 -12757.602} C_VEL
LIN {X 0,Y 368.887,Z 385.161,A -85,B 0,C 180,E1 -12761.102,E2 -12761.102} C_VEL
LIN {X 0,Y 368.913,Z 385.16,A -85,B 0,C 180,E1 -12764.532,E2 -12764.532} C_VEL
LIN {X 0,Y 369.044,Z 385.139,A -85,B 0,C 180,E1 -12766.79,E2 -12766.79} C_VEL
LIN {X 0,Y 369.046,Z 385.134,A -85,B 0,C 180,E1 -12770.131,E2 -12770.131} C_VEL
LIN {X 0,Y 369.137,Z 385.12,A -85,B 0,C 180,E1 -12773.441,E2 -12773.441} C_VEL
LIN {X 0,Y 369.291,Z 385.101,A -85,B 0,C 180,E1 -12777.819,E2 -12777.819} C_VEL
LIN {X 0,Y 369.289,Z 385.104,A -85,B 0,C 180,E1 -12782.182,E2 -12782.182} C_VEL
LIN {X 0,Y 369.154,Z 385.096,A -85,B 0,C 180,E1 -12786.671,E2 -12786.671} C_VEL
LIN {X 0,Y 369.048,Z 385.135,A -85,B 0,C 180,E1 -12789.869,E2 -12789.869} C_VEL
LIN {X 0,Y 369.026,Z 385.119,A -85,B 0,C 180,E1 -12793.773,E2 -12793.773} C_VEL
LIN {X 0,Y 368.98,Z 385.146,A -85,B 0,C 180,E1 -12797.744,E2 -12797.744} C_VEL
LIN {X 0,Y 368.898,Z 385.137,A -85,B 0,C 180,E1 -12801.222,E2 -12801.222} C_VEL
LIN {X 0,Y 368.906,Z 385.156,A -85,B 0,C 180,E1 -12803.877,E2 -12803.877} C_VEL
LIN {X 0,Y 368.848,Z 385.149,A -85,B 0,C 180,E1 -12807.213,E2 -12807.213} C_VEL
LIN {X 0,Y 368.884,Z 385.162,A -85,B 0,C 180,E1 -12809.693,E2 -12809.693} C_VEL
LIN {X 0,Y 368.887,Z 385.152,A -85,B 0,C 180,E1 -12813.044,E2 -12813.044} C_VEL
LIN {X 0,Y 368.904,Z 385.15,A -85,B 0,C 180,E1 -12816.199,E2 -12816.199} C_VEL
LIN {X 0,Y 368.867,Z 385.165,A -85,B 0,C 180,E1 -12818.958,E2 -12818.958} C_VEL
LIN {X 0,Y 368.864,Z 385.162,A -85,B 0,C 180,E1 -12822.009,E2 -12822.009} C_VEL
LIN {X 0,Y 368.871,Z 385.161,A -85,B 0,C 180,E1 -12825.176,E2 -12825.176} C_VEL
LIN {X 0,Y 368.887,Z 385.158,A -85,B 0,C 180,E1 -12828.86,E2 -12828.86} C_VEL
LIN {X 0,Y 368.882,Z 385.157,A -85,B 0,C 180,E1 -12829.057,E2 -12829.057} C_VEL
LIN {X 0,Y 369.899,Z 388.054,A -85,B 0,C 180,E1 -12829.248,E2 -12829.248} C_VEL
LIN {X 0,Y 371.519,Z 390.425,A -85,B 0,C 180,E1 -12829.484,E2 -12829.484} C_VEL
LIN {X 0,Y 379.949,Z 404.645,A -85,B 0,C 180,E1 -12830.714,E2 -12830.714} C_VEL
LIN {X 0,Y 389.041,Z 421.648,A -85,B 0,C 180,E1 -12831.993,E2 -12831.993} C_VEL
LIN {X 0,Y 386.95,Z 509.373,A -85,B 0,C 180,E1 -12833.683,E2 -12833.683} C_VEL
LIN {X 0,Y 386.643,Z 525.435,A -85,B 0,C 180,E1 -12834.113,E2 -12834.113} C_VEL
LIN {X 0,Y 386.028,Z 539.336,A -85,B 0,C 180,E1 -12834.679,E2 -12834.679} C_VEL
LIN {X 0,Y 385.017,Z 553.53,A -85,B 0,C 180,E1 -12835.451,E2 -12835.451} C_VEL
LIN {X 0,Y 383.867,Z 566.634,A -85,B 0,C 180,E1 -12836.371,E2 -12836.371} C_VEL
LIN {X 0,Y 382.497,Z 579.516,A -85,B 0,C 180,E1 -12837.492,E2 -12837.492} C_VEL
LIN {X 0,Y 380.794,Z 591.607,A -85,B 0,C 180,E1 -12838.753,E2 -12838.753} C_VEL
LIN {X 0,Y 379.158,Z 603.245,A -85,B 0,C 180,E1 -12840.24,E2 -12840.24} C_VEL
LIN {X 0,Y 377.318,Z 614.374,A -85,B 0,C 180,E1 -12841.947,E2 -12841.947} C_VEL
LIN {X 0,Y 375.633,Z 624.207,A -85,B 0,C 180,E1 -12843.774,E2 -12843.774} C_VEL
LIN {X 0,Y 374.138,Z 632.367,A -85,B 0,C 180,E1 -12845.591,E2 -12845.591} C_VEL
LIN {X 0,Y 372.789,Z 639.417,A -85,B 0,C 180,E1 -12847.485,E2 -12847.485} C_VEL
LIN {X 0,Y 371.667,Z 645.572,A -85,B 0,C 180,E1 -12849.524,E2 -12849.524} C_VEL
LIN {X 0,Y 370.778,Z 650.126,A -85,B 0,C 180,E1 -12851.395,E2 -12851.395} C_VEL
LIN {X 0,Y 370.05,Z 654.038,A -85,B 0,C 180,E1 -12853.449,E2 -12853.449} C_VEL
LIN {X 0,Y 369.467,Z 657.081,A -85,B 0,C 180,E1 -12855.684,E2 -12855.684} C_VEL
LIN {X 0,Y 369.109,Z 658.899,A -85,B 0,C 180,E1 -12857.911,E2 -12857.911} C_VEL
LIN {X 0,Y 368.984,Z 659.566,A -85,B 0,C 180,E1 -12860.13,E2 -12860.13} C_VEL
LIN {X 0,Y 368.989,Z 659.136,A -85,B 0,C 180,E1 -12862.339,E2 -12862.339} C_VEL
LIN {X 0,Y 369.036,Z 657.63,A -85,B 0,C 180,E1 -12864.537,E2 -12864.537} C_VEL
LIN {X 0,Y 369.356,Z 654.988,A -85,B 0,C 180,E1 -12866.728,E2 -12866.728} C_VEL
LIN {X 0,Y 369.724,Z 651.176,A -85,B 0,C 180,E1 -12868.911,E2 -12868.911} C_VEL
LIN {X 0,Y 370.38,Z 646.064,A -85,B 0,C 180,E1 -12871.088,E2 -12871.088} C_VEL
LIN {X 0,Y 371.36,Z 639.55,A -85,B 0,C 180,E1 -12873.255,E2 -12873.255} C_VEL
LIN {X 0,Y 372.415,Z 631.488,A -85,B 0,C 180,E1 -12875.415,E2 -12875.415} C_VEL
LIN {X 0,Y 373.621,Z 622.867,A -85,B 0,C 180,E1 -12877.295,E2 -12877.295} C_VEL
LIN {X 0,Y 374.864,Z 614.085,A -85,B 0,C 180,E1 -12878.898,E2 -12878.898} C_VEL
LIN {X 0,Y 376.159,Z 603.771,A -85,B 0,C 180,E1 -12880.496,E2 -12880.496} C_VEL
LIN {X 0,Y 377.508,Z 591.436,A -85,B 0,C 180,E1 -12882.09,E2 -12882.09} C_VEL
LIN {X 0,Y 378.879,Z 578.965,A -85,B 0,C 180,E1 -12883.407,E2 -12883.407} C_VEL
LIN {X 0,Y 379.011,Z 577.813,A -85,B 0,C 180,E1 -12883.516,E2 -12883.516} C_VEL
LIN {X 0,Y 378.928,Z 572.88,A -85,B 0,C 180,E1 -12884.006,E2 -12884.006} C_VEL
LIN {X 0,Y 377.007,Z 564.86,A -85,B 0,C 180,E1 -12884.845,E2 -12884.845} C_VEL
LIN {X 0,Y 375.06,Z 556.589,A -85,B 0,C 180,E1 -12885.62,E2 -12885.62} C_VEL
LIN {X 0,Y 374.814,Z 551.249,A -85,B 0,C 180,E1 -12885.999,E2 -12885.999} C_VEL
LIN {X 0,Y 375.661,Z 536.286,A -85,B 0,C 180,E1 -12886.782,E2 -12886.782} C_VEL
LIN {X 0,Y 376.095,Z 520.785,A -85,B 0,C 180,E1 -12887.365,E2 -12887.365} C_VEL
LIN {X 0,Y 376.381,Z 500.332,A -85,B 0,C 180,E1 -12887.831,E2 -12887.831} C_VEL
LIN {X 0,Y 378.142,Z 420.592,A -85,B 0,C 180,E1 -12889.358,E2 -12889.358} C_VEL
LIN {X 0,Y 371.557,Z 406.128,A -85,B 0,C 180,E1 -12890.171,E2 -12890.171} C_VEL
LIN {X 0,Y 363.155,Z 389.315,A -85,B 0,C 180,E1 -12891.223,E2 -12891.223} C_VEL
LIN {X 0,Y 361.993,Z 386.725,A -85,B 0,C 180,E1 -12891.379,E2 -12891.379} C_VEL
LIN {X 0,Y 361.862,Z 386.035,A -85,B 0,C 180,E1 -12891.441,E2 -12891.441} C_VEL
LIN {X 0,Y 361.852,Z 386.039,A -85,B 0,C 180,E1 -12895.296,E2 -12895.296} C_VEL
LIN {X 0,Y 361.837,Z 386.028,A -85,B 0,C 180,E1 -12899.068,E2 -12899.068} C_VEL
LIN {X 0,Y 361.837,Z 386.038,A -85,B 0,C 180,E1 -12901.629,E2 -12901.629} C_VEL
LIN {X 0,Y 361.869,Z 386.036,A -85,B 0,C 180,E1 -12905.343,E2 -12905.343} C_VEL
LIN {X 0,Y 361.823,Z 386.04,A -85,B 0,C 180,E1 -12909.017,E2 -12909.017} C_VEL
LIN {X 0,Y 361.81,Z 386.041,A -85,B 0,C 180,E1 -12912.832,E2 -12912.832} C_VEL
LIN {X 0,Y 361.806,Z 386.04,A -85,B 0,C 180,E1 -12915.948,E2 -12915.948} C_VEL
LIN {X 0,Y 361.807,Z 386.044,A -85,B 0,C 180,E1 -12919.249,E2 -12919.249} C_VEL
LIN {X 0,Y 361.857,Z 386.033,A -85,B 0,C 180,E1 -12922.98,E2 -12922.98} C_VEL
LIN {X 0,Y 361.853,Z 386.027,A -85,B 0,C 180,E1 -12926.631,E2 -12926.631} C_VEL
LIN {X 0,Y 361.842,Z 386.035,A -85,B 0,C 180,E1 -12929.669,E2 -12929.669} C_VEL
LIN {X 0,Y 361.848,Z 386.039,A -85,B 0,C 180,E1 -12933.466,E2 -12933.466} C_VEL
LIN {X 0,Y 361.868,Z 386.029,A -85,B 0,C 180,E1 -12937.143,E2 -12937.143} C_VEL
LIN {X 0,Y 361.877,Z 386.027,A -85,B 0,C 180,E1 -12940.721,E2 -12940.721} C_VEL
LIN {X 0,Y 361.934,Z 386.023,A -85,B 0,C 180,E1 -12944.225,E2 -12944.225} C_VEL
LIN {X 0,Y 361.993,Z 386.006,A -85,B 0,C 180,E1 -12946.527,E2 -12946.527} C_VEL
LIN {X 0,Y 361.988,Z 385.982,A -85,B 0,C 180,E1 -12949.936,E2 -12949.936} C_VEL
LIN {X 0,Y 362.11,Z 385.999,A -85,B 0,C 180,E1 -12953.312,E2 -12953.312} C_VEL
LIN {X 0,Y 362.246,Z 385.975,A -85,B 0,C 180,E1 -12957.776,E2 -12957.776} C_VEL
LIN {X 0,Y 362.258,Z 385.979,A -85,B 0,C 180,E1 -12962.223,E2 -12962.223} C_VEL
LIN {X 0,Y 362.1,Z 386.002,A -85,B 0,C 180,E1 -12966.687,E2 -12966.687} C_VEL
LIN {X 0,Y 361.989,Z 386.014,A -85,B 0,C 180,E1 -12970.063,E2 -12970.063} C_VEL
LIN {X 0,Y 361.973,Z 386.014,A -85,B 0,C 180,E1 -12973.887,E2 -12973.887} C_VEL
LIN {X 0,Y 361.87,Z 386.028,A -85,B 0,C 180,E1 -12978.104,E2 -12978.104} C_VEL
LIN {X 0,Y 361.846,Z 386.038,A -85,B 0,C 180,E1 -12981.656,E2 -12981.656} C_VEL
LIN {X 0,Y 361.845,Z 386.038,A -85,B 0,C 180,E1 -12985.296,E2 -12985.296} C_VEL
LIN {X 0,Y 361.849,Z 386.035,A -85,B 0,C 180,E1 -12989.074,E2 -12989.074} C_VEL
LIN {X 0,Y 361.841,Z 386.029,A -85,B 0,C 180,E1 -12992.945,E2 -12992.945} C_VEL
LIN {X 0,Y 361.857,Z 386.036,A -85,B 0,C 180,E1 -12995.638,E2 -12995.638} C_VEL
LIN {X 0,Y 361.819,Z 386.03,A -85,B 0,C 180,E1 -12999.018,E2 -12999.018} C_VEL
LIN {X 0,Y 361.824,Z 386.032,A -85,B 0,C 180,E1 -13002.83,E2 -13002.83} C_VEL
LIN {X 0,Y 361.808,Z 386.037,A -85,B 0,C 180,E1 -13005.948,E2 -13005.948} C_VEL
LIN {X 0,Y 361.838,Z 386.068,A -85,B 0,C 180,E1 -13009.244,E2 -13009.244} C_VEL
LIN {X 0,Y 366.408,Z 402.073,A -85,B 0,C 180,E1 -13012.297,E2 -13012.297} C_VEL
LIN {X 0,Y 370.336,Z 417.417,A -85,B 0,C 180,E1 -13015.041,E2 -13015.041} C_VEL
LIN {X 0,Y 371.608,Z 422.776,A -85,B 0,C 180,E1 -13015.962,E2 -13015.962} C_VEL
LIN {X 0,Y 371.31,Z 427.75,A -85,B 0,C 180,E1 -13016.709,E2 -13016.709} C_VEL
LIN {X 0,Y 369.405,Z 446.686,A -85,B 0,C 180,E1 -13019.461,E2 -13019.461} C_VEL
LIN {X 0,Y 377.061,Z 505.068,A -85,B 0,C 180,E1 -13021.249,E2 -13021.249} C_VEL
LIN {X 0,Y 374.639,Z 614.568,A -85,B 0,C 180,E1 -13023.355,E2 -13023.355} C_VEL
LIN {X 0,Y 373.816,Z 629.753,A -85,B 0,C 180,E1 -13023.818,E2 -13023.818} C_VEL
LIN {X 0,Y 372.521,Z 645.315,A -85,B 0,C 180,E1 -13024.508,E2 -13024.508} C_VEL
LIN {X 0,Y 370.972,Z 659.736,A -85,B 0,C 180,E1 -13025.368,E2 -13025.368} C_VEL
